   instPopulateLED.requests.row[148].pbSelection.animate := 255;
   instPopulateLED.requests.row[148].rtBackground.animate := 255;
   instPopulateLED.requests.row[148].tfDropZone.animate := 255;
   instPopulateLED.requests.row[148].tfDropZone.value := WSTRING#'';
   instPopulateLED.requests.row[148].tfLine.animate := 255;
   instPopulateLED.requests.row[148].tfLine.value := WSTRING#'';
   instPopulateLED.requests.row[148].tfPartNumber.animateDL := 255;
   instPopulateLED.requests.row[148].tfPartNumber.animateSL := 255;
   instPopulateLED.requests.row[148].tfPartNumber.value := WSTRING#'';
   instPopulateLED.requests.row[148].tfTime.animate := 255;
   instPopulateLED.requests.row[148].tfTime.value := WSTRING#'';
   instPopulateLED.requests.row[149].pbSelection.animate := 255;
   instPopulateLED.requests.row[149].rtBackground.animate := 255;
   instPopulateLED.requests.row[149].tfDropZone.animate := 255;
   instPopulateLED.requests.row[149].tfDropZone.value := WSTRING#'';
   instPopulateLED.requests.row[149].tfLine.animate := 255;
   instPopulateLED.requests.row[149].tfLine.value := WSTRING#'';
   instPopulateLED.requests.row[149].tfPartNumber.animateDL := 255;
   instPopulateLED.requests.row[149].tfPartNumber.animateSL := 255;
   instPopulateLED.requests.row[149].tfPartNumber.value := WSTRING#'';
   instPopulateLED.requests.row[149].tfTime.animate := 255;
   instPopulateLED.requests.row[149].tfTime.value := WSTRING#'';
   instPopulateLED.requests.row[150].pbSelection.animate := 255;
   instPopulateLED.requests.row[150].rtBackground.animate := 255;
   instPopulateLED.requests.row[150].tfDropZone.animate := 255;
   instPopulateLED.requests.row[150].tfDropZone.value := WSTRING#'';
   instPopulateLED.requests.row[150].tfLine.animate := 255;
   instPopulateLED.requests.row[150].tfLine.value := WSTRING#'';
   instPopulateLED.requests.row[150].tfPartNumber.animateDL := 255;
   instPopulateLED.requests.row[150].tfPartNumber.animateSL := 255;
   instPopulateLED.requests.row[150].tfPartNumber.value := WSTRING#'';
   instPopulateLED.requests.row[150].tfTime.animate := 255;
   instPopulateLED.requests.row[150].tfTime.value := WSTRING#'';
   instPopulateLED.requests.row[151].pbSelection.animate := 255;
   instPopulateLED.requests.row[151].rtBackground.animate := 255;
   instPopulateLED.requests.row[151].tfDropZone.animate := 255;
   instPopulateLED.requests.row[151].tfDropZone.value := WSTRING#'';
   instPopulateLED.requests.row[151].tfLine.animate := 255;
   instPopulateLED.requests.row[151].tfLine.value := WSTRING#'';
   instPopulateLED.requests.row[151].tfPartNumber.animateDL := 255;
   instPopulateLED.requests.row[151].tfPartNumber.animateSL := 255;
   instPopulateLED.requests.row[151].tfPartNumber.value := WSTRING#'';
   instPopulateLED.requests.row[151].tfTime.animate := 255;
   instPopulateLED.requests.row[151].tfTime.value := WSTRING#'';
   instPopulateLED.requests.row[152].pbSelection.animate := 255;
   instPopulateLED.requests.row[152].rtBackground.animate := 255;
   instPopulateLED.requests.row[152].tfDropZone.animate := 255;
   instPopulateLED.requests.row[152].tfDropZone.value := WSTRING#'';
   instPopulateLED.requests.row[152].tfLine.animate := 255;
   instPopulateLED.requests.row[152].tfLine.value := WSTRING#'';
   instPopulateLED.requests.row[152].tfPartNumber.animateDL := 255;
   instPopulateLED.requests.row[152].tfPartNumber.animateSL := 255;
   instPopulateLED.requests.row[152].tfPartNumber.value := WSTRING#'';
   instPopulateLED.requests.row[152].tfTime.animate := 255;
   instPopulateLED.requests.row[152].tfTime.value := WSTRING#'';
   instPopulateLED.requests.row[153].pbSelection.animate := 255;
   instPopulateLED.requests.row[153].rtBackground.animate := 255;
   instPopulateLED.requests.row[153].tfDropZone.animate := 255;
   instPopulateLED.requests.row[153].tfDropZone.value := WSTRING#'';
   instPopulateLED.requests.row[153].tfLine.animate := 255;
   instPopulateLED.requests.row[153].tfLine.value := WSTRING#'';
   instPopulateLED.requests.row[153].tfPartNumber.animateDL := 255;
   instPopulateLED.requests.row[153].tfPartNumber.animateSL := 255;
   instPopulateLED.requests.row[153].tfPartNumber.value := WSTRING#'';
   instPopulateLED.requests.row[153].tfTime.animate := 255;
   instPopulateLED.requests.row[153].tfTime.value := WSTRING#'';
   instPopulateLED.requests.row[154].pbSelection.animate := 255;
   instPopulateLED.requests.row[154].rtBackground.animate := 255;
   instPopulateLED.requests.row[154].tfDropZone.animate := 255;
   instPopulateLED.requests.row[154].tfDropZone.value := WSTRING#'';
   instPopulateLED.requests.row[154].tfLine.animate := 255;
   instPopulateLED.requests.row[154].tfLine.value := WSTRING#'';
   instPopulateLED.requests.row[154].tfPartNumber.animateDL := 255;
   instPopulateLED.requests.row[154].tfPartNumber.animateSL := 255;
   instPopulateLED.requests.row[154].tfPartNumber.value := WSTRING#'';
   instPopulateLED.requests.row[154].tfTime.animate := 255;
   instPopulateLED.requests.row[154].tfTime.value := WSTRING#'';
   instPopulateLED.requests.row[155].pbSelection.animate := 255;
   instPopulateLED.requests.row[155].rtBackground.animate := 255;
   instPopulateLED.requests.row[155].tfDropZone.animate := 255;
   instPopulateLED.requests.row[155].tfDropZone.value := WSTRING#'';
   instPopulateLED.requests.row[155].tfLine.animate := 255;
   instPopulateLED.requests.row[155].tfLine.value := WSTRING#'';
   instPopulateLED.requests.row[155].tfPartNumber.animateDL := 255;
   instPopulateLED.requests.row[155].tfPartNumber.animateSL := 255;
   instPopulateLED.requests.row[155].tfPartNumber.value := WSTRING#'';
   instPopulateLED.requests.row[155].tfTime.animate := 255;
   instPopulateLED.requests.row[155].tfTime.value := WSTRING#'';
   instPopulateLED.requests.row[156].pbSelection.animate := 255;
   instPopulateLED.requests.row[156].rtBackground.animate := 255;
   instPopulateLED.requests.row[156].tfDropZone.animate := 255;
   instPopulateLED.requests.row[156].tfDropZone.value := WSTRING#'';
   instPopulateLED.requests.row[156].tfLine.animate := 255;
   instPopulateLED.requests.row[156].tfLine.value := WSTRING#'';
   instPopulateLED.requests.row[156].tfPartNumber.animateDL := 255;
   instPopulateLED.requests.row[156].tfPartNumber.animateSL := 255;
   instPopulateLED.requests.row[156].tfPartNumber.value := WSTRING#'';
   instPopulateLED.requests.row[156].tfTime.animate := 255;
   instPopulateLED.requests.row[156].tfTime.value := WSTRING#'';
   instPopulateLED.requests.row[157].pbSelection.animate := 255;
   instPopulateLED.requests.row[157].rtBackground.animate := 255;
   instPopulateLED.requests.row[157].tfDropZone.animate := 255;
   instPopulateLED.requests.row[157].tfDropZone.value := WSTRING#'';
   instPopulateLED.requests.row[157].tfLine.animate := 255;
   instPopulateLED.requests.row[157].tfLine.value := WSTRING#'';
   instPopulateLED.requests.row[157].tfPartNumber.animateDL := 255;
   instPopulateLED.requests.row[157].tfPartNumber.animateSL := 255;
   instPopulateLED.requests.row[157].tfPartNumber.value := WSTRING#'';
   instPopulateLED.requests.row[157].tfTime.animate := 255;
   instPopulateLED.requests.row[157].tfTime.value := WSTRING#'';
   instPopulateLED.requests.row[158].pbSelection.animate := 255;
   instPopulateLED.requests.row[158].rtBackground.animate := 255;
   instPopulateLED.requests.row[158].tfDropZone.animate := 255;
   instPopulateLED.requests.row[158].tfDropZone.value := WSTRING#'';
   instPopulateLED.requests.row[158].tfLine.animate := 255;
   instPopulateLED.requests.row[158].tfLine.value := WSTRING#'';
   instPopulateLED.requests.row[158].tfPartNumber.animateDL := 255;
   instPopulateLED.requests.row[158].tfPartNumber.animateSL := 255;
   instPopulateLED.requests.row[158].tfPartNumber.value := WSTRING#'';
   instPopulateLED.requests.row[158].tfTime.animate := 255;
   instPopulateLED.requests.row[158].tfTime.value := WSTRING#'';
   instPopulateLED.requests.row[159].pbSelection.animate := 255;
   instPopulateLED.requests.row[159].rtBackground.animate := 255;
   instPopulateLED.requests.row[159].tfDropZone.animate := 255;
   instPopulateLED.requests.row[159].tfDropZone.value := WSTRING#'';
   instPopulateLED.requests.row[159].tfLine.animate := 255;
   instPopulateLED.requests.row[159].tfLine.value := WSTRING#'';
   instPopulateLED.requests.row[159].tfPartNumber.animateDL := 255;
   instPopulateLED.requests.row[159].tfPartNumber.animateSL := 255;
   instPopulateLED.requests.row[159].tfPartNumber.value := WSTRING#'';
   instPopulateLED.requests.row[159].tfTime.animate := 255;
   instPopulateLED.requests.row[159].tfTime.value := WSTRING#'';
   instPopulateLED.requests.row[160].pbSelection.animate := 255;
   instPopulateLED.requests.row[160].rtBackground.animate := 255;
   instPopulateLED.requests.row[160].tfDropZone.animate := 255;
   instPopulateLED.requests.row[160].tfDropZone.value := WSTRING#'';
   instPopulateLED.requests.row[160].tfLine.animate := 255;
   instPopulateLED.requests.row[160].tfLine.value := WSTRING#'';
   instPopulateLED.requests.row[160].tfPartNumber.animateDL := 255;
   instPopulateLED.requests.row[160].tfPartNumber.animateSL := 255;
   instPopulateLED.requests.row[160].tfPartNumber.value := WSTRING#'';
   instPopulateLED.requests.row[160].tfTime.animate := 255;
   instPopulateLED.requests.row[160].tfTime.value := WSTRING#'';
   instPopulateLED.requests.row[161].pbSelection.animate := 255;
   instPopulateLED.requests.row[161].rtBackground.animate := 255;
   instPopulateLED.requests.row[161].tfDropZone.animate := 255;
   instPopulateLED.requests.row[161].tfDropZone.value := WSTRING#'';
   instPopulateLED.requests.row[161].tfLine.animate := 255;
   instPopulateLED.requests.row[161].tfLine.value := WSTRING#'';
   instPopulateLED.requests.row[161].tfPartNumber.animateDL := 255;
   instPopulateLED.requests.row[161].tfPartNumber.animateSL := 255;
   instPopulateLED.requests.row[161].tfPartNumber.value := WSTRING#'';
   instPopulateLED.requests.row[161].tfTime.animate := 255;
   instPopulateLED.requests.row[161].tfTime.value := WSTRING#'';
   instPopulateLED.requests.row[162].pbSelection.animate := 255;
   instPopulateLED.requests.row[162].rtBackground.animate := 255;
   instPopulateLED.requests.row[162].tfDropZone.animate := 255;
   instPopulateLED.requests.row[162].tfDropZone.value := WSTRING#'';
   instPopulateLED.requests.row[162].tfLine.animate := 255;
   instPopulateLED.requests.row[162].tfLine.value := WSTRING#'';
   instPopulateLED.requests.row[162].tfPartNumber.animateDL := 255;
   instPopulateLED.requests.row[162].tfPartNumber.animateSL := 255;
   instPopulateLED.requests.row[162].tfPartNumber.value := WSTRING#'';
   instPopulateLED.requests.row[162].tfTime.animate := 255;
   instPopulateLED.requests.row[162].tfTime.value := WSTRING#'';
   instPopulateLED.requests.row[163].pbSelection.animate := 255;
   instPopulateLED.requests.row[163].rtBackground.animate := 255;
   instPopulateLED.requests.row[163].tfDropZone.animate := 255;
   instPopulateLED.requests.row[163].tfDropZone.value := WSTRING#'';
   instPopulateLED.requests.row[163].tfLine.animate := 255;
   instPopulateLED.requests.row[163].tfLine.value := WSTRING#'';
   instPopulateLED.requests.row[163].tfPartNumber.animateDL := 255;
   instPopulateLED.requests.row[163].tfPartNumber.animateSL := 255;
   instPopulateLED.requests.row[163].tfPartNumber.value := WSTRING#'';
   instPopulateLED.requests.row[163].tfTime.animate := 255;
   instPopulateLED.requests.row[163].tfTime.value := WSTRING#'';
   instPopulateLED.requests.row[164].pbSelection.animate := 255;
   instPopulateLED.requests.row[164].rtBackground.animate := 255;
   instPopulateLED.requests.row[164].tfDropZone.animate := 255;
   instPopulateLED.requests.row[164].tfDropZone.value := WSTRING#'';
   instPopulateLED.requests.row[164].tfLine.animate := 255;
   instPopulateLED.requests.row[164].tfLine.value := WSTRING#'';
   instPopulateLED.requests.row[164].tfPartNumber.animateDL := 255;
   instPopulateLED.requests.row[164].tfPartNumber.animateSL := 255;
   instPopulateLED.requests.row[164].tfPartNumber.value := WSTRING#'';
   instPopulateLED.requests.row[164].tfTime.animate := 255;
   instPopulateLED.requests.row[164].tfTime.value := WSTRING#'';
   instPopulateLED.requests.row[165].pbSelection.animate := 255;
   instPopulateLED.requests.row[165].rtBackground.animate := 255;
   instPopulateLED.requests.row[165].tfDropZone.animate := 255;
   instPopulateLED.requests.row[165].tfDropZone.value := WSTRING#'';
   instPopulateLED.requests.row[165].tfLine.animate := 255;
   instPopulateLED.requests.row[165].tfLine.value := WSTRING#'';
   instPopulateLED.requests.row[165].tfPartNumber.animateDL := 255;
   instPopulateLED.requests.row[165].tfPartNumber.animateSL := 255;
   instPopulateLED.requests.row[165].tfPartNumber.value := WSTRING#'';
   instPopulateLED.requests.row[165].tfTime.animate := 255;
   instPopulateLED.requests.row[165].tfTime.value := WSTRING#'';
   instPopulateLED.requests.row[166].pbSelection.animate := 255;
   instPopulateLED.requests.row[166].rtBackground.animate := 255;
   instPopulateLED.requests.row[166].tfDropZone.animate := 255;
   instPopulateLED.requests.row[166].tfDropZone.value := WSTRING#'';
   instPopulateLED.requests.row[166].tfLine.animate := 255;
   instPopulateLED.requests.row[166].tfLine.value := WSTRING#'';
   instPopulateLED.requests.row[166].tfPartNumber.animateDL := 255;
   instPopulateLED.requests.row[166].tfPartNumber.animateSL := 255;
   instPopulateLED.requests.row[166].tfPartNumber.value := WSTRING#'';
   instPopulateLED.requests.row[166].tfTime.animate := 255;
   instPopulateLED.requests.row[166].tfTime.value := WSTRING#'';
   instPopulateLED.requests.row[167].pbSelection.animate := 255;
   instPopulateLED.requests.row[167].rtBackground.animate := 255;
   instPopulateLED.requests.row[167].tfDropZone.animate := 255;
   instPopulateLED.requests.row[167].tfDropZone.value := WSTRING#'';
   instPopulateLED.requests.row[167].tfLine.animate := 255;
   instPopulateLED.requests.row[167].tfLine.value := WSTRING#'';
   instPopulateLED.requests.row[167].tfPartNumber.animateDL := 255;
   instPopulateLED.requests.row[167].tfPartNumber.animateSL := 255;
   instPopulateLED.requests.row[167].tfPartNumber.value := WSTRING#'';
   instPopulateLED.requests.row[167].tfTime.animate := 255;
   instPopulateLED.requests.row[167].tfTime.value := WSTRING#'';
   instPopulateLED.requests.row[168].pbSelection.animate := 255;
   instPopulateLED.requests.row[168].rtBackground.animate := 255;
   instPopulateLED.requests.row[168].tfDropZone.animate := 255;
   instPopulateLED.requests.row[168].tfDropZone.value := WSTRING#'';
   instPopulateLED.requests.row[168].tfLine.animate := 255;
   instPopulateLED.requests.row[168].tfLine.value := WSTRING#'';
   instPopulateLED.requests.row[168].tfPartNumber.animateDL := 255;
   instPopulateLED.requests.row[168].tfPartNumber.animateSL := 255;
   instPopulateLED.requests.row[168].tfPartNumber.value := WSTRING#'';
   instPopulateLED.requests.row[168].tfTime.animate := 255;
   instPopulateLED.requests.row[168].tfTime.value := WSTRING#'';
   instPopulateLED.requests.row[169].pbSelection.animate := 255;
   instPopulateLED.requests.row[169].rtBackground.animate := 255;
   instPopulateLED.requests.row[169].tfDropZone.animate := 255;
   instPopulateLED.requests.row[169].tfDropZone.value := WSTRING#'';
   instPopulateLED.requests.row[169].tfLine.animate := 255;
   instPopulateLED.requests.row[169].tfLine.value := WSTRING#'';
   instPopulateLED.requests.row[169].tfPartNumber.animateDL := 255;
   instPopulateLED.requests.row[169].tfPartNumber.animateSL := 255;
   instPopulateLED.requests.row[169].tfPartNumber.value := WSTRING#'';
   instPopulateLED.requests.row[169].tfTime.animate := 255;
   instPopulateLED.requests.row[169].tfTime.value := WSTRING#'';
   instPopulateLED.requests.row[170].pbSelection.animate := 255;
   instPopulateLED.requests.row[170].rtBackground.animate := 255;
   instPopulateLED.requests.row[170].tfDropZone.animate := 255;
   instPopulateLED.requests.row[170].tfDropZone.value := WSTRING#'';
   instPopulateLED.requests.row[170].tfLine.animate := 255;
   instPopulateLED.requests.row[170].tfLine.value := WSTRING#'';
   instPopulateLED.requests.row[170].tfPartNumber.animateDL := 255;
   instPopulateLED.requests.row[170].tfPartNumber.animateSL := 255;
   instPopulateLED.requests.row[170].tfPartNumber.value := WSTRING#'';
   instPopulateLED.requests.row[170].tfTime.animate := 255;
   instPopulateLED.requests.row[170].tfTime.value := WSTRING#'';
   instPopulateLED.requests.row[171].pbSelection.animate := 255;
   instPopulateLED.requests.row[171].rtBackground.animate := 255;
   instPopulateLED.requests.row[171].tfDropZone.animate := 255;
   instPopulateLED.requests.row[171].tfDropZone.value := WSTRING#'';
   instPopulateLED.requests.row[171].tfLine.animate := 255;
   instPopulateLED.requests.row[171].tfLine.value := WSTRING#'';
   instPopulateLED.requests.row[171].tfPartNumber.animateDL := 255;
   instPopulateLED.requests.row[171].tfPartNumber.animateSL := 255;
   instPopulateLED.requests.row[171].tfPartNumber.value := WSTRING#'';
   instPopulateLED.requests.row[171].tfTime.animate := 255;
   instPopulateLED.requests.row[171].tfTime.value := WSTRING#'';
   instPopulateLED.requests.row[172].pbSelection.animate := 255;
   instPopulateLED.requests.row[172].rtBackground.animate := 255;
   instPopulateLED.requests.row[172].tfDropZone.animate := 255;
   instPopulateLED.requests.row[172].tfDropZone.value := WSTRING#'';
   instPopulateLED.requests.row[172].tfLine.animate := 255;
   instPopulateLED.requests.row[172].tfLine.value := WSTRING#'';
   instPopulateLED.requests.row[172].tfPartNumber.animateDL := 255;
   instPopulateLED.requests.row[172].tfPartNumber.animateSL := 255;
   instPopulateLED.requests.row[172].tfPartNumber.value := WSTRING#'';
   instPopulateLED.requests.row[172].tfTime.animate := 255;
   instPopulateLED.requests.row[172].tfTime.value := WSTRING#'';
   instPopulateLED.requests.row[173].pbSelection.animate := 255;
   instPopulateLED.requests.row[173].rtBackground.animate := 255;
   instPopulateLED.requests.row[173].tfDropZone.animate := 255;
   instPopulateLED.requests.row[173].tfDropZone.value := WSTRING#'';
   instPopulateLED.requests.row[173].tfLine.animate := 255;
   instPopulateLED.requests.row[173].tfLine.value := WSTRING#'';
   instPopulateLED.requests.row[173].tfPartNumber.animateDL := 255;
   instPopulateLED.requests.row[173].tfPartNumber.animateSL := 255;
   instPopulateLED.requests.row[173].tfPartNumber.value := WSTRING#'';
   instPopulateLED.requests.row[173].tfTime.animate := 255;
   instPopulateLED.requests.row[173].tfTime.value := WSTRING#'';
   instPopulateLED.requests.row[174].pbSelection.animate := 255;
   instPopulateLED.requests.row[174].rtBackground.animate := 255;
   instPopulateLED.requests.row[174].tfDropZone.animate := 255;
   instPopulateLED.requests.row[174].tfDropZone.value := WSTRING#'';
   instPopulateLED.requests.row[174].tfLine.animate := 255;
   instPopulateLED.requests.row[174].tfLine.value := WSTRING#'';
   instPopulateLED.requests.row[174].tfPartNumber.animateDL := 255;
   instPopulateLED.requests.row[174].tfPartNumber.animateSL := 255;
   instPopulateLED.requests.row[174].tfPartNumber.value := WSTRING#'';
   instPopulateLED.requests.row[174].tfTime.animate := 255;
   instPopulateLED.requests.row[174].tfTime.value := WSTRING#'';
   instPopulateLED.requests.row[175].pbSelection.animate := 255;
   instPopulateLED.requests.row[175].rtBackground.animate := 255;
   instPopulateLED.requests.row[175].tfDropZone.animate := 255;
   instPopulateLED.requests.row[175].tfDropZone.value := WSTRING#'';
   instPopulateLED.requests.row[175].tfLine.animate := 255;
   instPopulateLED.requests.row[175].tfLine.value := WSTRING#'';
   instPopulateLED.requests.row[175].tfPartNumber.animateDL := 255;
   instPopulateLED.requests.row[175].tfPartNumber.animateSL := 255;
   instPopulateLED.requests.row[175].tfPartNumber.value := WSTRING#'';
   instPopulateLED.requests.row[175].tfTime.animate := 255;
   instPopulateLED.requests.row[175].tfTime.value := WSTRING#'';
   instPopulateLED.requests.row[176].pbSelection.animate := 255;
   instPopulateLED.requests.row[176].rtBackground.animate := 255;
   instPopulateLED.requests.row[176].tfDropZone.animate := 255;
   instPopulateLED.requests.row[176].tfDropZone.value := WSTRING#'';
   instPopulateLED.requests.row[176].tfLine.animate := 255;
   instPopulateLED.requests.row[176].tfLine.value := WSTRING#'';
   instPopulateLED.requests.row[176].tfPartNumber.animateDL := 255;
   instPopulateLED.requests.row[176].tfPartNumber.animateSL := 255;
   instPopulateLED.requests.row[176].tfPartNumber.value := WSTRING#'';
   instPopulateLED.requests.row[176].tfTime.animate := 255;
   instPopulateLED.requests.row[176].tfTime.value := WSTRING#'';
   instPopulateLED.requests.row[177].pbSelection.animate := 255;
   instPopulateLED.requests.row[177].rtBackground.animate := 255;
   instPopulateLED.requests.row[177].tfDropZone.animate := 255;
   instPopulateLED.requests.row[177].tfDropZone.value := WSTRING#'';
   instPopulateLED.requests.row[177].tfLine.animate := 255;
   instPopulateLED.requests.row[177].tfLine.value := WSTRING#'';
   instPopulateLED.requests.row[177].tfPartNumber.animateDL := 255;
   instPopulateLED.requests.row[177].tfPartNumber.animateSL := 255;
   instPopulateLED.requests.row[177].tfPartNumber.value := WSTRING#'';
   instPopulateLED.requests.row[177].tfTime.animate := 255;
   instPopulateLED.requests.row[177].tfTime.value := WSTRING#'';
   instPopulateLED.requests.row[178].pbSelection.animate := 255;
   instPopulateLED.requests.row[178].rtBackground.animate := 255;
   instPopulateLED.requests.row[178].tfDropZone.animate := 255;
   instPopulateLED.requests.row[178].tfDropZone.value := WSTRING#'';
   instPopulateLED.requests.row[178].tfLine.animate := 255;
   instPopulateLED.requests.row[178].tfLine.value := WSTRING#'';
   instPopulateLED.requests.row[178].tfPartNumber.animateDL := 255;
   instPopulateLED.requests.row[178].tfPartNumber.animateSL := 255;
   instPopulateLED.requests.row[178].tfPartNumber.value := WSTRING#'';
   instPopulateLED.requests.row[178].tfTime.animate := 255;
   instPopulateLED.requests.row[178].tfTime.value := WSTRING#'';
   instPopulateLED.requests.row[179].pbSelection.animate := 255;
   instPopulateLED.requests.row[179].rtBackground.animate := 255;
   instPopulateLED.requests.row[179].tfDropZone.animate := 255;
   instPopulateLED.requests.row[179].tfDropZone.value := WSTRING#'';
   instPopulateLED.requests.row[179].tfLine.animate := 255;
   instPopulateLED.requests.row[179].tfLine.value := WSTRING#'';
   instPopulateLED.requests.row[179].tfPartNumber.animateDL := 255;
   instPopulateLED.requests.row[179].tfPartNumber.animateSL := 255;
   instPopulateLED.requests.row[179].tfPartNumber.value := WSTRING#'';
   instPopulateLED.requests.row[179].tfTime.animate := 255;
   instPopulateLED.requests.row[179].tfTime.value := WSTRING#'';
   instPopulateLED.requests.row[180].pbSelection.animate := 255;
   instPopulateLED.requests.row[180].rtBackground.animate := 255;
   instPopulateLED.requests.row[180].tfDropZone.animate := 255;
   instPopulateLED.requests.row[180].tfDropZone.value := WSTRING#'';
   instPopulateLED.requests.row[180].tfLine.animate := 255;
   instPopulateLED.requests.row[180].tfLine.value := WSTRING#'';
   instPopulateLED.requests.row[180].tfPartNumber.animateDL := 255;
   instPopulateLED.requests.row[180].tfPartNumber.animateSL := 255;
   instPopulateLED.requests.row[180].tfPartNumber.value := WSTRING#'';
   instPopulateLED.requests.row[180].tfTime.animate := 255;
   instPopulateLED.requests.row[180].tfTime.value := WSTRING#'';
   instPopulateLED.requests.row[181].pbSelection.animate := 255;
   instPopulateLED.requests.row[181].rtBackground.animate := 255;
   instPopulateLED.requests.row[181].tfDropZone.animate := 255;
   instPopulateLED.requests.row[181].tfDropZone.value := WSTRING#'';
   instPopulateLED.requests.row[181].tfLine.animate := 255;
   instPopulateLED.requests.row[181].tfLine.value := WSTRING#'';
   instPopulateLED.requests.row[181].tfPartNumber.animateDL := 255;
   instPopulateLED.requests.row[181].tfPartNumber.animateSL := 255;
   instPopulateLED.requests.row[181].tfPartNumber.value := WSTRING#'';
   instPopulateLED.requests.row[181].tfTime.animate := 255;
   instPopulateLED.requests.row[181].tfTime.value := WSTRING#'';
   instPopulateLED.requests.row[182].pbSelection.animate := 255;
   instPopulateLED.requests.row[182].rtBackground.animate := 255;
   instPopulateLED.requests.row[182].tfDropZone.animate := 255;
   instPopulateLED.requests.row[182].tfDropZone.value := WSTRING#'';
   instPopulateLED.requests.row[182].tfLine.animate := 255;
   instPopulateLED.requests.row[182].tfLine.value := WSTRING#'';
   instPopulateLED.requests.row[182].tfPartNumber.animateDL := 255;
   instPopulateLED.requests.row[182].tfPartNumber.animateSL := 255;
   instPopulateLED.requests.row[182].tfPartNumber.value := WSTRING#'';
   instPopulateLED.requests.row[182].tfTime.animate := 255;
   instPopulateLED.requests.row[182].tfTime.value := WSTRING#'';
   instPopulateLED.requests.row[183].pbSelection.animate := 255;
   instPopulateLED.requests.row[183].rtBackground.animate := 255;
   instPopulateLED.requests.row[183].tfDropZone.animate := 255;
   instPopulateLED.requests.row[183].tfDropZone.value := WSTRING#'';
   instPopulateLED.requests.row[183].tfLine.animate := 255;
   instPopulateLED.requests.row[183].tfLine.value := WSTRING#'';
   instPopulateLED.requests.row[183].tfPartNumber.animateDL := 255;
   instPopulateLED.requests.row[183].tfPartNumber.animateSL := 255;
   instPopulateLED.requests.row[183].tfPartNumber.value := WSTRING#'';
   instPopulateLED.requests.row[183].tfTime.animate := 255;
   instPopulateLED.requests.row[183].tfTime.value := WSTRING#'';
   instPopulateLED.requests.row[184].pbSelection.animate := 255;
   instPopulateLED.requests.row[184].rtBackground.animate := 255;
   instPopulateLED.requests.row[184].tfDropZone.animate := 255;
   instPopulateLED.requests.row[184].tfDropZone.value := WSTRING#'';
   instPopulateLED.requests.row[184].tfLine.animate := 255;
   instPopulateLED.requests.row[184].tfLine.value := WSTRING#'';
   instPopulateLED.requests.row[184].tfPartNumber.animateDL := 255;
   instPopulateLED.requests.row[184].tfPartNumber.animateSL := 255;
   instPopulateLED.requests.row[184].tfPartNumber.value := WSTRING#'';
   instPopulateLED.requests.row[184].tfTime.animate := 255;
   instPopulateLED.requests.row[184].tfTime.value := WSTRING#'';
   instPopulateLED.requests.row[185].pbSelection.animate := 255;
   instPopulateLED.requests.row[185].rtBackground.animate := 255;
   instPopulateLED.requests.row[185].tfDropZone.animate := 255;
   instPopulateLED.requests.row[185].tfDropZone.value := WSTRING#'';
   instPopulateLED.requests.row[185].tfLine.animate := 255;
   instPopulateLED.requests.row[185].tfLine.value := WSTRING#'';
   instPopulateLED.requests.row[185].tfPartNumber.animateDL := 255;
   instPopulateLED.requests.row[185].tfPartNumber.animateSL := 255;
   instPopulateLED.requests.row[185].tfPartNumber.value := WSTRING#'';
   instPopulateLED.requests.row[185].tfTime.animate := 255;
   instPopulateLED.requests.row[185].tfTime.value := WSTRING#'';
   instPopulateLED.requests.row[186].pbSelection.animate := 255;
   instPopulateLED.requests.row[186].rtBackground.animate := 255;
   instPopulateLED.requests.row[186].tfDropZone.animate := 255;
   instPopulateLED.requests.row[186].tfDropZone.value := WSTRING#'';
   instPopulateLED.requests.row[186].tfLine.animate := 255;
   instPopulateLED.requests.row[186].tfLine.value := WSTRING#'';
   instPopulateLED.requests.row[186].tfPartNumber.animateDL := 255;
   instPopulateLED.requests.row[186].tfPartNumber.animateSL := 255;
   instPopulateLED.requests.row[186].tfPartNumber.value := WSTRING#'';
   instPopulateLED.requests.row[186].tfTime.animate := 255;
   instPopulateLED.requests.row[186].tfTime.value := WSTRING#'';
   instPopulateLED.requests.row[187].pbSelection.animate := 255;
   instPopulateLED.requests.row[187].rtBackground.animate := 255;
   instPopulateLED.requests.row[187].tfDropZone.animate := 255;
   instPopulateLED.requests.row[187].tfDropZone.value := WSTRING#'';
   instPopulateLED.requests.row[187].tfLine.animate := 255;
   instPopulateLED.requests.row[187].tfLine.value := WSTRING#'';
   instPopulateLED.requests.row[187].tfPartNumber.animateDL := 255;
   instPopulateLED.requests.row[187].tfPartNumber.animateSL := 255;
   instPopulateLED.requests.row[187].tfPartNumber.value := WSTRING#'';
   instPopulateLED.requests.row[187].tfTime.animate := 255;
   instPopulateLED.requests.row[187].tfTime.value := WSTRING#'';
   instPopulateLED.requests.row[188].pbSelection.animate := 255;
   instPopulateLED.requests.row[188].rtBackground.animate := 255;
   instPopulateLED.requests.row[188].tfDropZone.animate := 255;
   instPopulateLED.requests.row[188].tfDropZone.value := WSTRING#'';
   instPopulateLED.requests.row[188].tfLine.animate := 255;
   instPopulateLED.requests.row[188].tfLine.value := WSTRING#'';
   instPopulateLED.requests.row[188].tfPartNumber.animateDL := 255;
   instPopulateLED.requests.row[188].tfPartNumber.animateSL := 255;
   instPopulateLED.requests.row[188].tfPartNumber.value := WSTRING#'';
   instPopulateLED.requests.row[188].tfTime.animate := 255;
   instPopulateLED.requests.row[188].tfTime.value := WSTRING#'';
   instPopulateLED.requests.row[189].pbSelection.animate := 255;
   instPopulateLED.requests.row[189].rtBackground.animate := 255;
   instPopulateLED.requests.row[189].tfDropZone.animate := 255;
   instPopulateLED.requests.row[189].tfDropZone.value := WSTRING#'';
   instPopulateLED.requests.row[189].tfLine.animate := 255;
   instPopulateLED.requests.row[189].tfLine.value := WSTRING#'';
   instPopulateLED.requests.row[189].tfPartNumber.animateDL := 255;
   instPopulateLED.requests.row[189].tfPartNumber.animateSL := 255;
   instPopulateLED.requests.row[189].tfPartNumber.value := WSTRING#'';
   instPopulateLED.requests.row[189].tfTime.animate := 255;
   instPopulateLED.requests.row[189].tfTime.value := WSTRING#'';
   instPopulateLED.requests.row[190].pbSelection.animate := 255;
   instPopulateLED.requests.row[190].rtBackground.animate := 255;
   instPopulateLED.requests.row[190].tfDropZone.animate := 255;
   instPopulateLED.requests.row[190].tfDropZone.value := WSTRING#'';
   instPopulateLED.requests.row[190].tfLine.animate := 255;
   instPopulateLED.requests.row[190].tfLine.value := WSTRING#'';
   instPopulateLED.requests.row[190].tfPartNumber.animateDL := 255;
   instPopulateLED.requests.row[190].tfPartNumber.animateSL := 255;
   instPopulateLED.requests.row[190].tfPartNumber.value := WSTRING#'';
   instPopulateLED.requests.row[190].tfTime.animate := 255;
   instPopulateLED.requests.row[190].tfTime.value := WSTRING#'';
   instPopulateLED.requests.row[191].pbSelection.animate := 255;
   instPopulateLED.requests.row[191].rtBackground.animate := 255;
   instPopulateLED.requests.row[191].tfDropZone.animate := 255;
   instPopulateLED.requests.row[191].tfDropZone.value := WSTRING#'';
   instPopulateLED.requests.row[191].tfLine.animate := 255;
   instPopulateLED.requests.row[191].tfLine.value := WSTRING#'';
   instPopulateLED.requests.row[191].tfPartNumber.animateDL := 255;
   instPopulateLED.requests.row[191].tfPartNumber.animateSL := 255;
   instPopulateLED.requests.row[191].tfPartNumber.value := WSTRING#'';
   instPopulateLED.requests.row[191].tfTime.animate := 255;
   instPopulateLED.requests.row[191].tfTime.value := WSTRING#'';
   instPopulateLED.requests.row[192].pbSelection.animate := 255;
   instPopulateLED.requests.row[192].rtBackground.animate := 255;
   instPopulateLED.requests.row[192].tfDropZone.animate := 255;
   instPopulateLED.requests.row[192].tfDropZone.value := WSTRING#'';
   instPopulateLED.requests.row[192].tfLine.animate := 255;
   instPopulateLED.requests.row[192].tfLine.value := WSTRING#'';
   instPopulateLED.requests.row[192].tfPartNumber.animateDL := 255;
   instPopulateLED.requests.row[192].tfPartNumber.animateSL := 255;
   instPopulateLED.requests.row[192].tfPartNumber.value := WSTRING#'';
   instPopulateLED.requests.row[192].tfTime.animate := 255;
   instPopulateLED.requests.row[192].tfTime.value := WSTRING#'';
   instPopulateLED.requests.row[193].pbSelection.animate := 255;
   instPopulateLED.requests.row[193].rtBackground.animate := 255;
   instPopulateLED.requests.row[193].tfDropZone.animate := 255;
   instPopulateLED.requests.row[193].tfDropZone.value := WSTRING#'';
   instPopulateLED.requests.row[193].tfLine.animate := 255;
   instPopulateLED.requests.row[193].tfLine.value := WSTRING#'';
   instPopulateLED.requests.row[193].tfPartNumber.animateDL := 255;
   instPopulateLED.requests.row[193].tfPartNumber.animateSL := 255;
   instPopulateLED.requests.row[193].tfPartNumber.value := WSTRING#'';
   instPopulateLED.requests.row[193].tfTime.animate := 255;
   instPopulateLED.requests.row[193].tfTime.value := WSTRING#'';
   instPopulateLED.requests.row[194].pbSelection.animate := 255;
   instPopulateLED.requests.row[194].rtBackground.animate := 255;
   instPopulateLED.requests.row[194].tfDropZone.animate := 255;
   instPopulateLED.requests.row[194].tfDropZone.value := WSTRING#'';
   instPopulateLED.requests.row[194].tfLine.animate := 255;
   instPopulateLED.requests.row[194].tfLine.value := WSTRING#'';
   instPopulateLED.requests.row[194].tfPartNumber.animateDL := 255;
   instPopulateLED.requests.row[194].tfPartNumber.animateSL := 255;
   instPopulateLED.requests.row[194].tfPartNumber.value := WSTRING#'';
   instPopulateLED.requests.row[194].tfTime.animate := 255;
   instPopulateLED.requests.row[194].tfTime.value := WSTRING#'';
   instPopulateLED.requests.row[195].pbSelection.animate := 255;
   instPopulateLED.requests.row[195].rtBackground.animate := 255;
   instPopulateLED.requests.row[195].tfDropZone.animate := 255;
   instPopulateLED.requests.row[195].tfDropZone.value := WSTRING#'';
   instPopulateLED.requests.row[195].tfLine.animate := 255;
   instPopulateLED.requests.row[195].tfLine.value := WSTRING#'';
   instPopulateLED.requests.row[195].tfPartNumber.animateDL := 255;
   instPopulateLED.requests.row[195].tfPartNumber.animateSL := 255;
   instPopulateLED.requests.row[195].tfPartNumber.value := WSTRING#'';
   instPopulateLED.requests.row[195].tfTime.animate := 255;
   instPopulateLED.requests.row[195].tfTime.value := WSTRING#'';
   instPopulateLED.requests.row[196].pbSelection.animate := 255;
   instPopulateLED.requests.row[196].rtBackground.animate := 255;
   instPopulateLED.requests.row[196].tfDropZone.animate := 255;
   instPopulateLED.requests.row[196].tfDropZone.value := WSTRING#'';
   instPopulateLED.requests.row[196].tfLine.animate := 255;
   instPopulateLED.requests.row[196].tfLine.value := WSTRING#'';
   instPopulateLED.requests.row[196].tfPartNumber.animateDL := 255;
   instPopulateLED.requests.row[196].tfPartNumber.animateSL := 255;
   instPopulateLED.requests.row[196].tfPartNumber.value := WSTRING#'';
   instPopulateLED.requests.row[196].tfTime.animate := 255;
   instPopulateLED.requests.row[196].tfTime.value := WSTRING#'';
   instPopulateLED.requests.row[197].pbSelection.animate := 255;
   instPopulateLED.requests.row[197].rtBackground.animate := 255;
   instPopulateLED.requests.row[197].tfDropZone.animate := 255;
   instPopulateLED.requests.row[197].tfDropZone.value := WSTRING#'';
   instPopulateLED.requests.row[197].tfLine.animate := 255;
   instPopulateLED.requests.row[197].tfLine.value := WSTRING#'';
   instPopulateLED.requests.row[197].tfPartNumber.animateDL := 255;
   instPopulateLED.requests.row[197].tfPartNumber.animateSL := 255;
   instPopulateLED.requests.row[197].tfPartNumber.value := WSTRING#'';
   instPopulateLED.requests.row[197].tfTime.animate := 255;
   instPopulateLED.requests.row[197].tfTime.value := WSTRING#'';
   instPopulateLED.requests.row[198].pbSelection.animate := 255;
   instPopulateLED.requests.row[198].rtBackground.animate := 255;
   instPopulateLED.requests.row[198].tfDropZone.animate := 255;
   instPopulateLED.requests.row[198].tfDropZone.value := WSTRING#'';
   instPopulateLED.requests.row[198].tfLine.animate := 255;
   instPopulateLED.requests.row[198].tfLine.value := WSTRING#'';
   instPopulateLED.requests.row[198].tfPartNumber.animateDL := 255;
   instPopulateLED.requests.row[198].tfPartNumber.animateSL := 255;
   instPopulateLED.requests.row[198].tfPartNumber.value := WSTRING#'';
   instPopulateLED.requests.row[198].tfTime.animate := 255;
   instPopulateLED.requests.row[198].tfTime.value := WSTRING#'';
   instPopulateLED.requests.row[199].pbSelection.animate := 255;
   instPopulateLED.requests.row[199].rtBackground.animate := 255;
   instPopulateLED.requests.row[199].tfDropZone.animate := 255;
   instPopulateLED.requests.row[199].tfDropZone.value := WSTRING#'';
   instPopulateLED.requests.row[199].tfLine.animate := 255;
   instPopulateLED.requests.row[199].tfLine.value := WSTRING#'';
   instPopulateLED.requests.row[199].tfPartNumber.animateDL := 255;
   instPopulateLED.requests.row[199].tfPartNumber.animateSL := 255;
   instPopulateLED.requests.row[199].tfPartNumber.value := WSTRING#'';
   instPopulateLED.requests.row[199].tfTime.animate := 255;
   instPopulateLED.requests.row[199].tfTime.value := WSTRING#'';
   instRcrdPartReq.pRow := 6;
   instRcrdPartReq.old.presses.me[26,3] := TRUE;
   instRmvPartReq.pRow := 6;
   instRmvPartReq.old.partReq.me[26,3] := TRUE;
   stations.me[0].kp8Config.activate[3] := TRUE;
   stations.me[0].kp8Config.activate[7] := TRUE;
   stations.me[0].kp8Config.colorOn1[0] := 'off';
   stations.me[0].kp8Config.colorOn1[1] := 'off';
   stations.me[0].kp8Config.colorOn1[2] := 'off';
   stations.me[0].kp8Config.colorOn1[3] := 'yellow';
   stations.me[0].kp8Config.colorOn1[4] := 'off';
   stations.me[0].kp8Config.colorOn1[5] := 'off';
   stations.me[0].kp8Config.colorOn1[6] := 'off';
   stations.me[0].kp8Config.colorOn1[7] := 'yellow';
   stations.me[0].kp8Config.colorOn2[0] := 'off';
   stations.me[0].kp8Config.colorOn2[1] := 'off';
   stations.me[0].kp8Config.colorOn2[2] := 'off';
   stations.me[0].kp8Config.colorOn2[4] := 'off';
   stations.me[0].kp8Config.colorOn2[5] := 'off';
   stations.me[0].kp8Config.colorOn2[6] := 'off';
   stations.me[0].kp8Config.colorOff[0] := 'off';
   stations.me[0].kp8Config.colorOff[1] := 'off';
   stations.me[0].kp8Config.colorOff[2] := 'off';
   stations.me[0].kp8Config.colorOff[3] := 'green';
   stations.me[0].kp8Config.colorOff[4] := 'off';
   stations.me[0].kp8Config.colorOff[5] := 'off';
   stations.me[0].kp8Config.colorOff[6] := 'off';
   stations.me[0].kp8Config.colorOff[7] := 'green';
   stations.me[0].kp8Config.mode[3] := TRUE;
   stations.me[0].kp8Config.mode[7] := TRUE;
   stations.me[0].kp8Out := 16#0088_0000;
   stations.me[0].presetTime.allotted[3] := 1800.0;
   stations.me[0].presetTime.allotted[7] := 1800.0;
   stations.me[0].presetTime.critical[3] := 300.0;
   stations.me[0].presetTime.critical[7] := 300.0;
   stations.me[0].stackLightOut := 16#2400_0000;
   stations.me[1].kp8Config.activate[2] := TRUE;
   stations.me[1].kp8Config.activate[3] := TRUE;
   stations.me[1].kp8Config.activate[6] := TRUE;
   stations.me[1].kp8Config.activate[7] := TRUE;
   stations.me[1].kp8Config.colorOn1[0] := 'off';
   stations.me[1].kp8Config.colorOn1[1] := 'off';
   stations.me[1].kp8Config.colorOn1[2] := 'yellow';
   stations.me[1].kp8Config.colorOn1[3] := 'yellow';
   stations.me[1].kp8Config.colorOn1[4] := 'off';
   stations.me[1].kp8Config.colorOn1[5] := 'off';
   stations.me[1].kp8Config.colorOn1[6] := 'yellow';
   stations.me[1].kp8Config.colorOn1[7] := 'yellow';
   stations.me[1].kp8Config.colorOn2[0] := 'off';
   stations.me[1].kp8Config.colorOn2[1] := 'off';
   stations.me[1].kp8Config.colorOn2[4] := 'off';
   stations.me[1].kp8Config.colorOn2[5] := 'off';
   stations.me[1].kp8Config.colorOff[0] := 'off';
   stations.me[1].kp8Config.colorOff[1] := 'off';
   stations.me[1].kp8Config.colorOff[2] := 'green';
   stations.me[1].kp8Config.colorOff[3] := 'green';
   stations.me[1].kp8Config.colorOff[4] := 'off';
   stations.me[1].kp8Config.colorOff[5] := 'off';
   stations.me[1].kp8Config.colorOff[6] := 'green';
   stations.me[1].kp8Config.colorOff[7] := 'green';
   stations.me[1].kp8Config.mode[2] := TRUE;
   stations.me[1].kp8Config.mode[3] := TRUE;
   stations.me[1].kp8Config.mode[6] := TRUE;
   stations.me[1].kp8Config.mode[7] := TRUE;
   stations.me[1].kp8Out := 16#00CC_0000;
   stations.me[1].presetTime.allotted[2] := 1800.0;
   stations.me[1].presetTime.allotted[3] := 1800.0;
   stations.me[1].presetTime.allotted[6] := 1800.0;
   stations.me[1].presetTime.allotted[7] := 1800.0;
   stations.me[1].presetTime.critical[2] := 300.0;
   stations.me[1].presetTime.critical[3] := 300.0;
   stations.me[1].presetTime.critical[6] := 300.0;
   stations.me[1].presetTime.critical[7] := 300.0;
   stations.me[1].stackLightOut := 16#2409_0000;
   stations.me[2].kp8Config.activate[1] := TRUE;
   stations.me[2].kp8Config.activate[2] := TRUE;
   stations.me[2].kp8Config.activate[3] := TRUE;
   stations.me[2].kp8Config.activate[5] := TRUE;
   stations.me[2].kp8Config.activate[6] := TRUE;
   stations.me[2].kp8Config.activate[7] := TRUE;
   stations.me[2].kp8Config.colorOn1[0] := 'off';
   stations.me[2].kp8Config.colorOn1[1] := 'yellow';
   stations.me[2].kp8Config.colorOn1[2] := 'yellow';
   stations.me[2].kp8Config.colorOn1[3] := 'yellow';
   stations.me[2].kp8Config.colorOn1[4] := 'off';
   stations.me[2].kp8Config.colorOn1[5] := 'yellow';
   stations.me[2].kp8Config.colorOn1[6] := 'yellow';
   stations.me[2].kp8Config.colorOn1[7] := 'yellow';
   stations.me[2].kp8Config.colorOn2[0] := 'off';
   stations.me[2].kp8Config.colorOn2[4] := 'off';
   stations.me[2].kp8Config.colorOff[0] := 'off';
   stations.me[2].kp8Config.colorOff[1] := 'green';
   stations.me[2].kp8Config.colorOff[2] := 'green';
   stations.me[2].kp8Config.colorOff[3] := 'green';
   stations.me[2].kp8Config.colorOff[4] := 'off';
   stations.me[2].kp8Config.colorOff[5] := 'green';
   stations.me[2].kp8Config.colorOff[6] := 'green';
   stations.me[2].kp8Config.colorOff[7] := 'green';
   stations.me[2].kp8Config.mode[1] := TRUE;
   stations.me[2].kp8Config.mode[2] := TRUE;
   stations.me[2].kp8Config.mode[3] := TRUE;
   stations.me[2].kp8Config.mode[5] := TRUE;
   stations.me[2].kp8Config.mode[6] := TRUE;
   stations.me[2].kp8Config.mode[7] := TRUE;
   stations.me[2].kp8Out := 16#00EE_0000;
   stations.me[2].presetTime.allotted[1] := 1800.0;
   stations.me[2].presetTime.allotted[2] := 1800.0;
   stations.me[2].presetTime.allotted[3] := 1800.0;
   stations.me[2].presetTime.allotted[5] := 1800.0;
   stations.me[2].presetTime.allotted[6] := 1800.0;
   stations.me[2].presetTime.allotted[7] := 1800.0;
   stations.me[2].presetTime.critical[1] := 300.0;
   stations.me[2].presetTime.critical[2] := 300.0;
   stations.me[2].presetTime.critical[3] := 300.0;
   stations.me[2].presetTime.critical[5] := 300.0;
   stations.me[2].presetTime.critical[6] := 300.0;
   stations.me[2].presetTime.critical[7] := 300.0;
   stations.me[2].stackLightOut := 16#2449_0200;
   stations.me[3].kp8Config.activate[1] := TRUE;
   stations.me[3].kp8Config.activate[2] := TRUE;
   stations.me[3].kp8Config.activate[3] := TRUE;
   stations.me[3].kp8Config.activate[5] := TRUE;
   stations.me[3].kp8Config.activate[6] := TRUE;
   stations.me[3].kp8Config.activate[7] := TRUE;
   stations.me[3].kp8Config.colorOn1[0] := 'off';
   stations.me[3].kp8Config.colorOn1[1] := 'yellow';
   stations.me[3].kp8Config.colorOn1[2] := 'yellow';
   stations.me[3].kp8Config.colorOn1[3] := 'yellow';
   stations.me[3].kp8Config.colorOn1[4] := 'off';
   stations.me[3].kp8Config.colorOn1[5] := 'yellow';
   stations.me[3].kp8Config.colorOn1[6] := 'yellow';
   stations.me[3].kp8Config.colorOn1[7] := 'yellow';
   stations.me[3].kp8Config.colorOn2[0] := 'off';
   stations.me[3].kp8Config.colorOn2[4] := 'off';
   stations.me[3].kp8Config.colorOff[0] := 'off';
   stations.me[3].kp8Config.colorOff[1] := 'green';
   stations.me[3].kp8Config.colorOff[2] := 'green';
   stations.me[3].kp8Config.colorOff[3] := 'green';
   stations.me[3].kp8Config.colorOff[4] := 'off';
   stations.me[3].kp8Config.colorOff[5] := 'green';
   stations.me[3].kp8Config.colorOff[6] := 'green';
   stations.me[3].kp8Config.colorOff[7] := 'green';
   stations.me[3].kp8Config.mode[1] := TRUE;
   stations.me[3].kp8Config.mode[2] := TRUE;
   stations.me[3].kp8Config.mode[3] := TRUE;
   stations.me[3].kp8Config.mode[5] := TRUE;
   stations.me[3].kp8Config.mode[6] := TRUE;
   stations.me[3].kp8Config.mode[7] := TRUE;
   stations.me[3].kp8Out := 16#00EE_0000;
   stations.me[3].presetTime.allotted[1] := 1800.0;
   stations.me[3].presetTime.allotted[2] := 1800.0;
   stations.me[3].presetTime.allotted[3] := 1800.0;
   stations.me[3].presetTime.allotted[5] := 1800.0;
   stations.me[3].presetTime.allotted[6] := 1800.0;
   stations.me[3].presetTime.allotted[7] := 1800.0;
   stations.me[3].presetTime.critical[1] := 300.0;
   stations.me[3].presetTime.critical[2] := 300.0;
   stations.me[3].presetTime.critical[3] := 300.0;
   stations.me[3].presetTime.critical[5] := 300.0;
   stations.me[3].presetTime.critical[6] := 300.0;
   stations.me[3].presetTime.critical[7] := 300.0;
   stations.me[3].stackLightOut := 16#2449_0200;
   stations.me[4].kp8Config.activate[7] := TRUE;
   stations.me[4].kp8Config.colorOn1[0] := 'off';
   stations.me[4].kp8Config.colorOn1[1] := 'off';
   stations.me[4].kp8Config.colorOn1[2] := 'off';
   stations.me[4].kp8Config.colorOn1[3] := 'off';
   stations.me[4].kp8Config.colorOn1[4] := 'off';
   stations.me[4].kp8Config.colorOn1[5] := 'off';
   stations.me[4].kp8Config.colorOn1[6] := 'off';
   stations.me[4].kp8Config.colorOn1[7] := 'yellow';
   stations.me[4].kp8Config.colorOn2[0] := 'off';
   stations.me[4].kp8Config.colorOn2[1] := 'off';
   stations.me[4].kp8Config.colorOn2[2] := 'off';
   stations.me[4].kp8Config.colorOn2[3] := 'off';
   stations.me[4].kp8Config.colorOn2[4] := 'off';
   stations.me[4].kp8Config.colorOn2[5] := 'off';
   stations.me[4].kp8Config.colorOn2[6] := 'off';
   stations.me[4].kp8Config.colorOff[0] := 'off';
   stations.me[4].kp8Config.colorOff[1] := 'off';
   stations.me[4].kp8Config.colorOff[2] := 'off';
   stations.me[4].kp8Config.colorOff[3] := 'off';
   stations.me[4].kp8Config.colorOff[4] := 'off';
   stations.me[4].kp8Config.colorOff[5] := 'off';
   stations.me[4].kp8Config.colorOff[6] := 'off';
   stations.me[4].kp8Config.colorOff[7] := 'green';
   stations.me[4].kp8Config.mode[7] := TRUE;
   stations.me[4].kp8Out := 16#0080_0000;
   stations.me[4].presetTime.allotted[7] := 1800.0;
   stations.me[4].presetTime.critical[7] := 300.0;
   stations.me[4].stackLightOut := 16#0400_0000;
   stations.me[5].kp8Config.activate[1] := TRUE;
   stations.me[5].kp8Config.activate[2] := TRUE;
   stations.me[5].kp8Config.activate[3] := TRUE;
   stations.me[5].kp8Config.activate[5] := TRUE;
   stations.me[5].kp8Config.activate[6] := TRUE;
   stations.me[5].kp8Config.activate[7] := TRUE;
   stations.me[5].kp8Config.colorOn1[0] := 'off';
   stations.me[5].kp8Config.colorOn1[1] := 'yellow';
   stations.me[5].kp8Config.colorOn1[2] := 'yellow';
   stations.me[5].kp8Config.colorOn1[3] := 'yellow';
   stations.me[5].kp8Config.colorOn1[4] := 'off';
   stations.me[5].kp8Config.colorOn1[5] := 'yellow';
   stations.me[5].kp8Config.colorOn1[6] := 'yellow';
   stations.me[5].kp8Config.colorOn1[7] := 'yellow';
   stations.me[5].kp8Config.colorOn2[0] := 'off';
   stations.me[5].kp8Config.colorOn2[4] := 'off';
   stations.me[5].kp8Config.colorOff[0] := 'off';
   stations.me[5].kp8Config.colorOff[1] := 'green';
   stations.me[5].kp8Config.colorOff[2] := 'green';
   stations.me[5].kp8Config.colorOff[3] := 'green';
   stations.me[5].kp8Config.colorOff[4] := 'off';
   stations.me[5].kp8Config.colorOff[5] := 'green';
   stations.me[5].kp8Config.colorOff[6] := 'green';
   stations.me[5].kp8Config.colorOff[7] := 'green';
   stations.me[5].kp8Config.mode[1] := TRUE;
   stations.me[5].kp8Config.mode[2] := TRUE;
   stations.me[5].kp8Config.mode[3] := TRUE;
   stations.me[5].kp8Config.mode[5] := TRUE;
   stations.me[5].kp8Config.mode[6] := TRUE;
   stations.me[5].kp8Config.mode[7] := TRUE;
   stations.me[5].kp8Out := 16#00EE_0000;
   stations.me[5].presetTime.allotted[1] := 1800.0;
   stations.me[5].presetTime.allotted[2] := 1800.0;
   stations.me[5].presetTime.allotted[3] := 1800.0;
   stations.me[5].presetTime.allotted[5] := 1800.0;
   stations.me[5].presetTime.allotted[6] := 1800.0;
   stations.me[5].presetTime.allotted[7] := 1800.0;
   stations.me[5].presetTime.critical[1] := 300.0;
   stations.me[5].presetTime.critical[2] := 300.0;
   stations.me[5].presetTime.critical[3] := 300.0;
   stations.me[5].presetTime.critical[5] := 300.0;
   stations.me[5].presetTime.critical[6] := 300.0;
   stations.me[5].presetTime.critical[7] := 300.0;
   stations.me[5].stackLightOut := 16#2449_0200;
   stations.me[6].kp8Config.activate[1] := TRUE;
   stations.me[6].kp8Config.activate[2] := TRUE;
   stations.me[6].kp8Config.activate[3] := TRUE;
   stations.me[6].kp8Config.activate[5] := TRUE;
   stations.me[6].kp8Config.activate[6] := TRUE;
   stations.me[6].kp8Config.activate[7] := TRUE;
   stations.me[6].kp8Config.colorOn1[0] := 'off';
   stations.me[6].kp8Config.colorOn1[1] := 'yellow';
   stations.me[6].kp8Config.colorOn1[2] := 'yellow';
   stations.me[6].kp8Config.colorOn1[3] := 'yellow';
   stations.me[6].kp8Config.colorOn1[4] := 'off';
   stations.me[6].kp8Config.colorOn1[5] := 'yellow';
   stations.me[6].kp8Config.colorOn1[6] := 'yellow';
   stations.me[6].kp8Config.colorOn1[7] := 'yellow';
   stations.me[6].kp8Config.colorOn2[0] := 'off';
   stations.me[6].kp8Config.colorOn2[4] := 'off';
   stations.me[6].kp8Config.colorOff[0] := 'off';
   stations.me[6].kp8Config.colorOff[1] := 'green';
   stations.me[6].kp8Config.colorOff[2] := 'green';
   stations.me[6].kp8Config.colorOff[3] := 'green';
   stations.me[6].kp8Config.colorOff[4] := 'off';
   stations.me[6].kp8Config.colorOff[5] := 'green';
   stations.me[6].kp8Config.colorOff[6] := 'green';
   stations.me[6].kp8Config.colorOff[7] := 'green';
   stations.me[6].kp8Config.mode[1] := TRUE;
   stations.me[6].kp8Config.mode[2] := TRUE;
   stations.me[6].kp8Config.mode[3] := TRUE;
   stations.me[6].kp8Config.mode[5] := TRUE;
   stations.me[6].kp8Config.mode[6] := TRUE;
   stations.me[6].kp8Config.mode[7] := TRUE;
   stations.me[6].kp8Out := 16#00EE_0000;
   stations.me[6].presetTime.allotted[1] := 1800.0;
   stations.me[6].presetTime.allotted[2] := 1800.0;
   stations.me[6].presetTime.allotted[3] := 1800.0;
   stations.me[6].presetTime.allotted[5] := 1800.0;
   stations.me[6].presetTime.allotted[6] := 1800.0;
   stations.me[6].presetTime.allotted[7] := 1800.0;
   stations.me[6].presetTime.critical[1] := 300.0;
   stations.me[6].presetTime.critical[2] := 300.0;
   stations.me[6].presetTime.critical[3] := 300.0;
   stations.me[6].presetTime.critical[5] := 300.0;
   stations.me[6].presetTime.critical[6] := 300.0;
   stations.me[6].presetTime.critical[7] := 300.0;
   stations.me[6].stackLightOut := 16#2449_0200;
   stations.me[7].kp8Config.activate[3] := TRUE;
   stations.me[7].kp8Config.activate[6] := TRUE;
   stations.me[7].kp8Config.activate[7] := TRUE;
   stations.me[7].kp8Config.colorOn1[0] := 'off';
   stations.me[7].kp8Config.colorOn1[1] := 'off';
   stations.me[7].kp8Config.colorOn1[2] := 'off';
   stations.me[7].kp8Config.colorOn1[3] := 'yellow';
   stations.me[7].kp8Config.colorOn1[4] := 'off';
   stations.me[7].kp8Config.colorOn1[5] := 'off';
   stations.me[7].kp8Config.colorOn1[6] := 'yellow';
   stations.me[7].kp8Config.colorOn1[7] := 'yellow';
   stations.me[7].kp8Config.colorOn2[0] := 'off';
   stations.me[7].kp8Config.colorOn2[1] := 'off';
   stations.me[7].kp8Config.colorOn2[2] := 'off';
   stations.me[7].kp8Config.colorOn2[4] := 'off';
   stations.me[7].kp8Config.colorOn2[5] := 'off';
   stations.me[7].kp8Config.colorOff[0] := 'off';
   stations.me[7].kp8Config.colorOff[1] := 'off';
   stations.me[7].kp8Config.colorOff[2] := 'off';
   stations.me[7].kp8Config.colorOff[3] := 'green';
   stations.me[7].kp8Config.colorOff[4] := 'off';
   stations.me[7].kp8Config.colorOff[5] := 'off';
   stations.me[7].kp8Config.colorOff[6] := 'green';
   stations.me[7].kp8Config.colorOff[7] := 'green';
   stations.me[7].kp8Config.mode[3] := TRUE;
   stations.me[7].kp8Config.mode[6] := TRUE;
   stations.me[7].kp8Config.mode[7] := TRUE;
   stations.me[7].kp8Out := 16#00C8_0000;
   stations.me[7].presetTime.allotted[3] := 1800.0;
   stations.me[7].presetTime.allotted[6] := 1800.0;
   stations.me[7].presetTime.allotted[7] := 1800.0;
   stations.me[7].presetTime.critical[3] := 300.0;
   stations.me[7].presetTime.critical[6] := 300.0;
   stations.me[7].presetTime.critical[7] := 300.0;
   stations.me[7].settings.btnSelection[3] := TRUE;
   stations.me[7].stackLightOut := 16#2401_0000;
   stations.me[8].kp8Config.activate[3] := TRUE;
   stations.me[8].kp8Config.activate[6] := TRUE;
   stations.me[8].kp8Config.activate[7] := TRUE;
   stations.me[8].kp8Config.colorOn1[0] := 'off';
   stations.me[8].kp8Config.colorOn1[1] := 'off';
   stations.me[8].kp8Config.colorOn1[2] := 'off';
   stations.me[8].kp8Config.colorOn1[3] := 'yellow';
   stations.me[8].kp8Config.colorOn1[4] := 'off';
   stations.me[8].kp8Config.colorOn1[5] := 'off';
   stations.me[8].kp8Config.colorOn1[6] := 'yellow';
   stations.me[8].kp8Config.colorOn1[7] := 'yellow';
   stations.me[8].kp8Config.colorOn2[0] := 'off';
   stations.me[8].kp8Config.colorOn2[1] := 'off';
   stations.me[8].kp8Config.colorOn2[2] := 'off';
   stations.me[8].kp8Config.colorOn2[4] := 'off';
   stations.me[8].kp8Config.colorOn2[5] := 'off';
   stations.me[8].kp8Config.colorOff[0] := 'off';
   stations.me[8].kp8Config.colorOff[1] := 'off';
   stations.me[8].kp8Config.colorOff[2] := 'off';
   stations.me[8].kp8Config.colorOff[3] := 'green';
   stations.me[8].kp8Config.colorOff[4] := 'off';
   stations.me[8].kp8Config.colorOff[5] := 'off';
   stations.me[8].kp8Config.colorOff[6] := 'green';
   stations.me[8].kp8Config.colorOff[7] := 'green';
   stations.me[8].kp8Config.mode[3] := TRUE;
   stations.me[8].kp8Config.mode[6] := TRUE;
   stations.me[8].kp8Config.mode[7] := TRUE;
   stations.me[8].kp8Out := 16#00C8_0000;
   stations.me[8].presetTime.allotted[3] := 1800.0;
   stations.me[8].presetTime.allotted[6] := 1800.0;
   stations.me[8].presetTime.allotted[7] := 1800.0;
   stations.me[8].presetTime.critical[3] := 300.0;
   stations.me[8].presetTime.critical[6] := 300.0;
   stations.me[8].presetTime.critical[7] := 300.0;
   stations.me[8].stackLightOut := 16#2401_0000;
   stations.me[9].kp8Config.activate[3] := TRUE;
   stations.me[9].kp8Config.activate[7] := TRUE;
   stations.me[9].kp8Config.colorOn1[0] := 'off';
   stations.me[9].kp8Config.colorOn1[1] := 'off';
   stations.me[9].kp8Config.colorOn1[2] := 'off';
   stations.me[9].kp8Config.colorOn1[3] := 'yellow';
   stations.me[9].kp8Config.colorOn1[4] := 'off';
   stations.me[9].kp8Config.colorOn1[5] := 'off';
   stations.me[9].kp8Config.colorOn1[6] := 'off';
   stations.me[9].kp8Config.colorOn1[7] := 'yellow';
   stations.me[9].kp8Config.colorOn2[0] := 'off';
   stations.me[9].kp8Config.colorOn2[1] := 'off';
   stations.me[9].kp8Config.colorOn2[2] := 'off';
   stations.me[9].kp8Config.colorOn2[4] := 'off';
   stations.me[9].kp8Config.colorOn2[5] := 'off';
   stations.me[9].kp8Config.colorOn2[6] := 'off';
   stations.me[9].kp8Config.colorOff[0] := 'off';
   stations.me[9].kp8Config.colorOff[1] := 'off';
   stations.me[9].kp8Config.colorOff[2] := 'off';
   stations.me[9].kp8Config.colorOff[3] := 'green';
   stations.me[9].kp8Config.colorOff[4] := 'off';
   stations.me[9].kp8Config.colorOff[5] := 'off';
   stations.me[9].kp8Config.colorOff[6] := 'off';
   stations.me[9].kp8Config.colorOff[7] := 'green';
   stations.me[9].kp8Config.mode[3] := TRUE;
   stations.me[9].kp8Config.mode[7] := TRUE;
   stations.me[9].kp8Out := 16#0088_0000;
   stations.me[9].presetTime.allotted[3] := 1800.0;
   stations.me[9].presetTime.allotted[7] := 1800.0;
   stations.me[9].presetTime.critical[3] := 300.0;
   stations.me[9].presetTime.critical[7] := 300.0;
   stations.me[9].stackLightOut := 16#2400_0000;
   stations.me[10].kp8Config.activate[3] := TRUE;
   stations.me[10].kp8Config.activate[6] := TRUE;
   stations.me[10].kp8Config.activate[7] := TRUE;
   stations.me[10].kp8Config.colorOn1[0] := 'off';
   stations.me[10].kp8Config.colorOn1[1] := 'off';
   stations.me[10].kp8Config.colorOn1[2] := 'off';
   stations.me[10].kp8Config.colorOn1[3] := 'yellow';
   stations.me[10].kp8Config.colorOn1[4] := 'off';
   stations.me[10].kp8Config.colorOn1[5] := 'off';
   stations.me[10].kp8Config.colorOn1[6] := 'yellow';
   stations.me[10].kp8Config.colorOn1[7] := 'yellow';
   stations.me[10].kp8Config.colorOn2[0] := 'off';
   stations.me[10].kp8Config.colorOn2[1] := 'off';
   stations.me[10].kp8Config.colorOn2[2] := 'off';
   stations.me[10].kp8Config.colorOn2[4] := 'off';
   stations.me[10].kp8Config.colorOn2[5] := 'off';
   stations.me[10].kp8Config.colorOff[0] := 'off';
   stations.me[10].kp8Config.colorOff[1] := 'off';
   stations.me[10].kp8Config.colorOff[2] := 'off';
   stations.me[10].kp8Config.colorOff[3] := 'green';
   stations.me[10].kp8Config.colorOff[4] := 'off';
   stations.me[10].kp8Config.colorOff[5] := 'off';
   stations.me[10].kp8Config.colorOff[6] := 'green';
   stations.me[10].kp8Config.colorOff[7] := 'green';
   stations.me[10].kp8Config.mode[3] := TRUE;
   stations.me[10].kp8Config.mode[6] := TRUE;
   stations.me[10].kp8Config.mode[7] := TRUE;
   stations.me[10].kp8Out := 16#00C8_0000;
   stations.me[10].presetTime.allotted[3] := 1800.0;
   stations.me[10].presetTime.allotted[6] := 1800.0;
   stations.me[10].presetTime.allotted[7] := 1800.0;
   stations.me[10].presetTime.critical[3] := 300.0;
   stations.me[10].presetTime.critical[6] := 300.0;
   stations.me[10].presetTime.critical[7] := 300.0;
   stations.me[10].stackLightOut := 16#2401_0000;
   stations.me[11].kp8Config.activate[3] := TRUE;
   stations.me[11].kp8Config.activate[6] := TRUE;
   stations.me[11].kp8Config.activate[7] := TRUE;
   stations.me[11].kp8Config.colorOn1[0] := 'off';
   stations.me[11].kp8Config.colorOn1[1] := 'off';
   stations.me[11].kp8Config.colorOn1[2] := 'off';
   stations.me[11].kp8Config.colorOn1[3] := 'yellow';
   stations.me[11].kp8Config.colorOn1[4] := 'off';
   stations.me[11].kp8Config.colorOn1[5] := 'off';
   stations.me[11].kp8Config.colorOn1[6] := 'yellow';
   stations.me[11].kp8Config.colorOn1[7] := 'yellow';
   stations.me[11].kp8Config.colorOn2[0] := 'off';
   stations.me[11].kp8Config.colorOn2[1] := 'off';
   stations.me[11].kp8Config.colorOn2[2] := 'off';
   stations.me[11].kp8Config.colorOn2[4] := 'off';
   stations.me[11].kp8Config.colorOn2[5] := 'off';
   stations.me[11].kp8Config.colorOff[0] := 'off';
   stations.me[11].kp8Config.colorOff[1] := 'off';
   stations.me[11].kp8Config.colorOff[2] := 'off';
   stations.me[11].kp8Config.colorOff[3] := 'green';
   stations.me[11].kp8Config.colorOff[4] := 'off';
   stations.me[11].kp8Config.colorOff[5] := 'off';
   stations.me[11].kp8Config.colorOff[6] := 'green';
   stations.me[11].kp8Config.colorOff[7] := 'green';
   stations.me[11].kp8Config.mode[3] := TRUE;
   stations.me[11].kp8Config.mode[6] := TRUE;
   stations.me[11].kp8Config.mode[7] := TRUE;
   stations.me[11].kp8Out := 16#00C8_0000;
   stations.me[11].presetTime.allotted[3] := 1800.0;
   stations.me[11].presetTime.allotted[6] := 1800.0;
   stations.me[11].presetTime.allotted[7] := 1800.0;
   stations.me[11].presetTime.critical[3] := 300.0;
   stations.me[11].presetTime.critical[6] := 300.0;
   stations.me[11].presetTime.critical[7] := 300.0;
   stations.me[11].stackLightOut := 16#2401_0000;
   stations.me[12].kp8Config.activate[1] := TRUE;
   stations.me[12].kp8Config.activate[2] := TRUE;
   stations.me[12].kp8Config.activate[3] := TRUE;
   stations.me[12].kp8Config.activate[5] := TRUE;
   stations.me[12].kp8Config.activate[6] := TRUE;
   stations.me[12].kp8Config.activate[7] := TRUE;
   stations.me[12].kp8Config.colorOn1[0] := 'off';
   stations.me[12].kp8Config.colorOn1[1] := 'yellow';
   stations.me[12].kp8Config.colorOn1[2] := 'yellow';
   stations.me[12].kp8Config.colorOn1[3] := 'yellow';
   stations.me[12].kp8Config.colorOn1[4] := 'off';
   stations.me[12].kp8Config.colorOn1[5] := 'yellow';
   stations.me[12].kp8Config.colorOn1[6] := 'yellow';
   stations.me[12].kp8Config.colorOn1[7] := 'yellow';
   stations.me[12].kp8Config.colorOn2[0] := 'off';
   stations.me[12].kp8Config.colorOn2[4] := 'off';
   stations.me[12].kp8Config.colorOff[0] := 'off';
   stations.me[12].kp8Config.colorOff[1] := 'green';
   stations.me[12].kp8Config.colorOff[2] := 'green';
   stations.me[12].kp8Config.colorOff[3] := 'green';
   stations.me[12].kp8Config.colorOff[4] := 'off';
   stations.me[12].kp8Config.colorOff[5] := 'green';
   stations.me[12].kp8Config.colorOff[6] := 'green';
   stations.me[12].kp8Config.colorOff[7] := 'green';
   stations.me[12].kp8Config.mode[1] := TRUE;
   stations.me[12].kp8Config.mode[2] := TRUE;
   stations.me[12].kp8Config.mode[3] := TRUE;
   stations.me[12].kp8Config.mode[5] := TRUE;
   stations.me[12].kp8Config.mode[6] := TRUE;
   stations.me[12].kp8Config.mode[7] := TRUE;
   stations.me[12].kp8Out := 16#00EE_0000;
   stations.me[12].presetTime.allotted[1] := 1800.0;
   stations.me[12].presetTime.allotted[2] := 1800.0;
   stations.me[12].presetTime.allotted[3] := 1800.0;
   stations.me[12].presetTime.allotted[5] := 1800.0;
   stations.me[12].presetTime.allotted[6] := 1800.0;
   stations.me[12].presetTime.allotted[7] := 1800.0;
   stations.me[12].presetTime.critical[1] := 300.0;
   stations.me[12].presetTime.critical[2] := 300.0;
   stations.me[12].presetTime.critical[3] := 300.0;
   stations.me[12].presetTime.critical[5] := 300.0;
   stations.me[12].presetTime.critical[6] := 300.0;
   stations.me[12].presetTime.critical[7] := 300.0;
   stations.me[12].stackLightOut := 16#2449_0200;
   stations.me[13].kp8Config.activate[2] := TRUE;
   stations.me[13].kp8Config.activate[3] := TRUE;
   stations.me[13].kp8Config.activate[6] := TRUE;
   stations.me[13].kp8Config.activate[7] := TRUE;
   stations.me[13].kp8Config.colorOn1[0] := 'off';
   stations.me[13].kp8Config.colorOn1[1] := 'off';
   stations.me[13].kp8Config.colorOn1[2] := 'yellow';
   stations.me[13].kp8Config.colorOn1[3] := 'yellow';
   stations.me[13].kp8Config.colorOn1[4] := 'off';
   stations.me[13].kp8Config.colorOn1[5] := 'off';
   stations.me[13].kp8Config.colorOn1[6] := 'yellow';
   stations.me[13].kp8Config.colorOn1[7] := 'yellow';
   stations.me[13].kp8Config.colorOn2[0] := 'off';
   stations.me[13].kp8Config.colorOn2[1] := 'off';
   stations.me[13].kp8Config.colorOn2[4] := 'off';
   stations.me[13].kp8Config.colorOn2[5] := 'off';
   stations.me[13].kp8Config.colorOff[0] := 'off';
   stations.me[13].kp8Config.colorOff[1] := 'off';
   stations.me[13].kp8Config.colorOff[2] := 'green';
   stations.me[13].kp8Config.colorOff[3] := 'green';
   stations.me[13].kp8Config.colorOff[4] := 'off';
   stations.me[13].kp8Config.colorOff[5] := 'off';
   stations.me[13].kp8Config.colorOff[6] := 'green';
   stations.me[13].kp8Config.colorOff[7] := 'green';
   stations.me[13].kp8Config.mode[2] := TRUE;
   stations.me[13].kp8Config.mode[3] := TRUE;
   stations.me[13].kp8Config.mode[6] := TRUE;
   stations.me[13].kp8Config.mode[7] := TRUE;
   stations.me[13].kp8Out := 16#00CC_0000;
   stations.me[13].presetTime.allotted[2] := 1800.0;
   stations.me[13].presetTime.allotted[3] := 1800.0;
   stations.me[13].presetTime.allotted[6] := 1800.0;
   stations.me[13].presetTime.allotted[7] := 1800.0;
   stations.me[13].presetTime.critical[2] := 300.0;
   stations.me[13].presetTime.critical[3] := 300.0;
   stations.me[13].presetTime.critical[6] := 300.0;
   stations.me[13].presetTime.critical[7] := 300.0;
   stations.me[13].stackLightOut := 16#2409_0000;
   stations.me[14].kp8Config.activate[2] := TRUE;
   stations.me[14].kp8Config.activate[3] := TRUE;
   stations.me[14].kp8Config.activate[5] := TRUE;
   stations.me[14].kp8Config.activate[6] := TRUE;
   stations.me[14].kp8Config.activate[7] := TRUE;
   stations.me[14].kp8Config.colorOn1[0] := 'off';
   stations.me[14].kp8Config.colorOn1[1] := 'off';
   stations.me[14].kp8Config.colorOn1[2] := 'yellow';
   stations.me[14].kp8Config.colorOn1[3] := 'yellow';
   stations.me[14].kp8Config.colorOn1[4] := 'off';
   stations.me[14].kp8Config.colorOn1[5] := 'yellow';
   stations.me[14].kp8Config.colorOn1[6] := 'yellow';
   stations.me[14].kp8Config.colorOn1[7] := 'yellow';
   stations.me[14].kp8Config.colorOn2[0] := 'off';
   stations.me[14].kp8Config.colorOn2[1] := 'off';
   stations.me[14].kp8Config.colorOn2[4] := 'off';
   stations.me[14].kp8Config.colorOff[0] := 'off';
   stations.me[14].kp8Config.colorOff[1] := 'off';
   stations.me[14].kp8Config.colorOff[2] := 'green';
   stations.me[14].kp8Config.colorOff[3] := 'green';
   stations.me[14].kp8Config.colorOff[4] := 'off';
   stations.me[14].kp8Config.colorOff[5] := 'green';
   stations.me[14].kp8Config.colorOff[6] := 'green';
   stations.me[14].kp8Config.colorOff[7] := 'green';
   stations.me[14].kp8Config.mode[2] := TRUE;
   stations.me[14].kp8Config.mode[3] := TRUE;
   stations.me[14].kp8Config.mode[5] := TRUE;
   stations.me[14].kp8Config.mode[6] := TRUE;
   stations.me[14].kp8Config.mode[7] := TRUE;
   stations.me[14].kp8Out := 16#00EC_0000;
   stations.me[14].presetTime.allotted[2] := 1800.0;
   stations.me[14].presetTime.allotted[3] := 1800.0;
   stations.me[14].presetTime.allotted[5] := 1800.0;
   stations.me[14].presetTime.allotted[6] := 1800.0;
   stations.me[14].presetTime.allotted[7] := 1800.0;
   stations.me[14].presetTime.critical[2] := 300.0;
   stations.me[14].presetTime.critical[3] := 300.0;
   stations.me[14].presetTime.critical[5] := 300.0;
   stations.me[14].presetTime.critical[6] := 300.0;
   stations.me[14].presetTime.critical[7] := 300.0;
   stations.me[14].stackLightOut := 16#2449_0000;
   stations.me[15].kp8Config.activate[1] := TRUE;
   stations.me[15].kp8Config.activate[2] := TRUE;
   stations.me[15].kp8Config.activate[3] := TRUE;
   stations.me[15].kp8Config.activate[5] := TRUE;
   stations.me[15].kp8Config.activate[6] := TRUE;
   stations.me[15].kp8Config.activate[7] := TRUE;
   stations.me[15].kp8Config.colorOn1[0] := 'off';
   stations.me[15].kp8Config.colorOn1[1] := 'yellow';
   stations.me[15].kp8Config.colorOn1[2] := 'yellow';
   stations.me[15].kp8Config.colorOn1[3] := 'yellow';
   stations.me[15].kp8Config.colorOn1[4] := 'off';
   stations.me[15].kp8Config.colorOn1[5] := 'yellow';
   stations.me[15].kp8Config.colorOn1[6] := 'yellow';
   stations.me[15].kp8Config.colorOn1[7] := 'yellow';
   stations.me[15].kp8Config.colorOn2[0] := 'off';
   stations.me[15].kp8Config.colorOn2[4] := 'off';
   stations.me[15].kp8Config.colorOff[0] := 'off';
   stations.me[15].kp8Config.colorOff[1] := 'green';
   stations.me[15].kp8Config.colorOff[2] := 'green';
   stations.me[15].kp8Config.colorOff[3] := 'green';
   stations.me[15].kp8Config.colorOff[4] := 'off';
   stations.me[15].kp8Config.colorOff[5] := 'green';
   stations.me[15].kp8Config.colorOff[6] := 'green';
   stations.me[15].kp8Config.colorOff[7] := 'green';
   stations.me[15].kp8Config.mode[1] := TRUE;
   stations.me[15].kp8Config.mode[2] := TRUE;
   stations.me[15].kp8Config.mode[3] := TRUE;
   stations.me[15].kp8Config.mode[5] := TRUE;
   stations.me[15].kp8Config.mode[6] := TRUE;
   stations.me[15].kp8Config.mode[7] := TRUE;
   stations.me[15].kp8Out := 16#00EE_0000;
   stations.me[15].presetTime.allotted[1] := 1800.0;
   stations.me[15].presetTime.allotted[2] := 1800.0;
   stations.me[15].presetTime.allotted[3] := 1800.0;
   stations.me[15].presetTime.allotted[5] := 1800.0;
   stations.me[15].presetTime.allotted[6] := 1800.0;
   stations.me[15].presetTime.allotted[7] := 1800.0;
   stations.me[15].presetTime.critical[1] := 300.0;
   stations.me[15].presetTime.critical[2] := 300.0;
   stations.me[15].presetTime.critical[3] := 300.0;
   stations.me[15].presetTime.critical[5] := 300.0;
   stations.me[15].presetTime.critical[6] := 300.0;
   stations.me[15].presetTime.critical[7] := 300.0;
   stations.me[15].stackLightOut := 16#2449_0200;
   stations.me[16].kp8Config.activate[3] := TRUE;
   stations.me[16].kp8Config.activate[7] := TRUE;
   stations.me[16].kp8Config.colorOn1[0] := 'off';
   stations.me[16].kp8Config.colorOn1[1] := 'off';
   stations.me[16].kp8Config.colorOn1[2] := 'off';
   stations.me[16].kp8Config.colorOn1[3] := 'yellow';
   stations.me[16].kp8Config.colorOn1[4] := 'off';
   stations.me[16].kp8Config.colorOn1[5] := 'off';
   stations.me[16].kp8Config.colorOn1[6] := 'off';
   stations.me[16].kp8Config.colorOn1[7] := 'yellow';
   stations.me[16].kp8Config.colorOn2[0] := 'off';
   stations.me[16].kp8Config.colorOn2[1] := 'off';
   stations.me[16].kp8Config.colorOn2[2] := 'off';
   stations.me[16].kp8Config.colorOn2[4] := 'off';
   stations.me[16].kp8Config.colorOn2[5] := 'off';
   stations.me[16].kp8Config.colorOn2[6] := 'off';
   stations.me[16].kp8Config.colorOff[0] := 'off';
   stations.me[16].kp8Config.colorOff[1] := 'off';
   stations.me[16].kp8Config.colorOff[2] := 'off';
   stations.me[16].kp8Config.colorOff[3] := 'green';
   stations.me[16].kp8Config.colorOff[4] := 'off';
   stations.me[16].kp8Config.colorOff[5] := 'off';
   stations.me[16].kp8Config.colorOff[6] := 'off';
   stations.me[16].kp8Config.colorOff[7] := 'green';
   stations.me[16].kp8Config.mode[3] := TRUE;
   stations.me[16].kp8Config.mode[7] := TRUE;
   stations.me[16].kp8Out := 16#0088_0000;
   stations.me[16].presetTime.allotted[3] := 1800.0;
   stations.me[16].presetTime.allotted[6] := 1800.0;
   stations.me[16].presetTime.allotted[7] := 1800.0;
   stations.me[16].presetTime.critical[3] := 300.0;
   stations.me[16].presetTime.critical[6] := 300.0;
   stations.me[16].presetTime.critical[7] := 300.0;
   stations.me[16].stackLightOut := 16#2400_0000;
   stations.me[17].kp8Config.activate[2] := TRUE;
   stations.me[17].kp8Config.activate[3] := TRUE;
   stations.me[17].kp8Config.activate[6] := TRUE;
   stations.me[17].kp8Config.activate[7] := TRUE;
   stations.me[17].kp8Config.colorOn1[0] := 'off';
   stations.me[17].kp8Config.colorOn1[1] := 'off';
   stations.me[17].kp8Config.colorOn1[2] := 'yellow';
   stations.me[17].kp8Config.colorOn1[3] := 'yellow';
   stations.me[17].kp8Config.colorOn1[4] := 'off';
   stations.me[17].kp8Config.colorOn1[5] := 'off';
   stations.me[17].kp8Config.colorOn1[6] := 'yellow';
   stations.me[17].kp8Config.colorOn1[7] := 'yellow';
   stations.me[17].kp8Config.colorOn2[0] := 'off';
   stations.me[17].kp8Config.colorOn2[1] := 'off';
   stations.me[17].kp8Config.colorOn2[4] := 'off';
   stations.me[17].kp8Config.colorOn2[5] := 'off';
   stations.me[17].kp8Config.colorOff[0] := 'off';
   stations.me[17].kp8Config.colorOff[1] := 'off';
   stations.me[17].kp8Config.colorOff[2] := 'green';
   stations.me[17].kp8Config.colorOff[3] := 'green';
   stations.me[17].kp8Config.colorOff[4] := 'off';
   stations.me[17].kp8Config.colorOff[5] := 'off';
   stations.me[17].kp8Config.colorOff[6] := 'green';
   stations.me[17].kp8Config.colorOff[7] := 'green';
   stations.me[17].kp8Config.mode[2] := TRUE;
   stations.me[17].kp8Config.mode[3] := TRUE;
   stations.me[17].kp8Config.mode[6] := TRUE;
   stations.me[17].kp8Config.mode[7] := TRUE;
   stations.me[17].kp8Out := 16#00CC_0000;
   stations.me[17].presetTime.allotted[2] := 1800.0;
   stations.me[17].presetTime.allotted[3] := 1800.0;
   stations.me[17].presetTime.allotted[6] := 1800.0;
   stations.me[17].presetTime.allotted[7] := 1800.0;
   stations.me[17].presetTime.critical[2] := 300.0;
   stations.me[17].presetTime.critical[3] := 300.0;
   stations.me[17].presetTime.critical[6] := 300.0;
   stations.me[17].presetTime.critical[7] := 300.0;
   stations.me[17].stackLightOut := 16#2409_0000;
   stations.me[18].kp8Config.activate[3] := TRUE;
   stations.me[18].kp8Config.activate[6] := TRUE;
   stations.me[18].kp8Config.activate[7] := TRUE;
   stations.me[18].kp8Config.colorOn1[0] := 'off';
   stations.me[18].kp8Config.colorOn1[1] := 'off';
   stations.me[18].kp8Config.colorOn1[2] := 'off';
   stations.me[18].kp8Config.colorOn1[3] := 'yellow';
   stations.me[18].kp8Config.colorOn1[4] := 'off';
   stations.me[18].kp8Config.colorOn1[5] := 'off';
   stations.me[18].kp8Config.colorOn1[6] := 'yellow';
   stations.me[18].kp8Config.colorOn1[7] := 'yellow';
   stations.me[18].kp8Config.colorOn2[0] := 'off';
   stations.me[18].kp8Config.colorOn2[1] := 'off';
   stations.me[18].kp8Config.colorOn2[2] := 'off';
   stations.me[18].kp8Config.colorOn2[4] := 'off';
   stations.me[18].kp8Config.colorOn2[5] := 'off';
   stations.me[18].kp8Config.colorOff[0] := 'off';
   stations.me[18].kp8Config.colorOff[1] := 'off';
   stations.me[18].kp8Config.colorOff[2] := 'off';
   stations.me[18].kp8Config.colorOff[3] := 'green';
   stations.me[18].kp8Config.colorOff[4] := 'off';
   stations.me[18].kp8Config.colorOff[5] := 'off';
   stations.me[18].kp8Config.colorOff[6] := 'green';
   stations.me[18].kp8Config.colorOff[7] := 'green';
   stations.me[18].kp8Config.mode[3] := TRUE;
   stations.me[18].kp8Config.mode[6] := TRUE;
   stations.me[18].kp8Config.mode[7] := TRUE;
   stations.me[18].kp8Out := 16#00C8_0000;
   stations.me[18].presetTime.allotted[3] := 1800.0;
   stations.me[18].presetTime.allotted[6] := 1800.0;
   stations.me[18].presetTime.allotted[7] := 1800.0;
   stations.me[18].presetTime.critical[3] := 300.0;
   stations.me[18].presetTime.critical[6] := 300.0;
   stations.me[18].presetTime.critical[7] := 300.0;
   stations.me[18].stackLightOut := 16#2401_0000;
   stations.me[19].kp8Config.activate[1] := TRUE;
   stations.me[19].kp8Config.activate[2] := TRUE;
   stations.me[19].kp8Config.activate[3] := TRUE;
   stations.me[19].kp8Config.activate[5] := TRUE;
   stations.me[19].kp8Config.activate[6] := TRUE;
   stations.me[19].kp8Config.activate[7] := TRUE;
   stations.me[19].kp8Config.colorOn1[0] := 'off';
   stations.me[19].kp8Config.colorOn1[1] := 'yellow';
   stations.me[19].kp8Config.colorOn1[2] := 'yellow';
   stations.me[19].kp8Config.colorOn1[3] := 'yellow';
   stations.me[19].kp8Config.colorOn1[4] := 'off';
   stations.me[19].kp8Config.colorOn1[5] := 'yellow';
   stations.me[19].kp8Config.colorOn1[6] := 'yellow';
   stations.me[19].kp8Config.colorOn1[7] := 'yellow';
   stations.me[19].kp8Config.colorOn2[0] := 'off';
   stations.me[19].kp8Config.colorOn2[4] := 'off';
   stations.me[19].kp8Config.colorOff[0] := 'off';
   stations.me[19].kp8Config.colorOff[1] := 'green';
   stations.me[19].kp8Config.colorOff[2] := 'green';
   stations.me[19].kp8Config.colorOff[3] := 'green';
   stations.me[19].kp8Config.colorOff[4] := 'off';
   stations.me[19].kp8Config.colorOff[5] := 'green';
   stations.me[19].kp8Config.colorOff[6] := 'green';
   stations.me[19].kp8Config.colorOff[7] := 'green';
   stations.me[19].kp8Config.mode[1] := TRUE;
   stations.me[19].kp8Config.mode[2] := TRUE;
   stations.me[19].kp8Config.mode[3] := TRUE;
   stations.me[19].kp8Config.mode[5] := TRUE;
   stations.me[19].kp8Config.mode[6] := TRUE;
   stations.me[19].kp8Config.mode[7] := TRUE;
   stations.me[19].kp8Out := 16#00EE_0000;
   stations.me[19].presetTime.allotted[1] := 1800.0;
   stations.me[19].presetTime.allotted[2] := 1800.0;
   stations.me[19].presetTime.allotted[3] := 1800.0;
   stations.me[19].presetTime.allotted[5] := 120.0;
   stations.me[19].presetTime.allotted[6] := 1800.0;
   stations.me[19].presetTime.allotted[7] := 1800.0;
   stations.me[19].presetTime.critical[1] := 300.0;
   stations.me[19].presetTime.critical[2] := 300.0;
   stations.me[19].presetTime.critical[3] := 300.0;
   stations.me[19].presetTime.critical[5] := 70.0;
   stations.me[19].presetTime.critical[6] := 300.0;
   stations.me[19].presetTime.critical[7] := 300.0;
   stations.me[19].settings.selected := TRUE;
   stations.me[19].stackLightOut := 16#2449_0200;
   stations.me[20].kp8Config.colorOn1[0] := 'off';
   stations.me[20].kp8Config.colorOn1[1] := 'off';
   stations.me[20].kp8Config.colorOn1[2] := 'off';
   stations.me[20].kp8Config.colorOn1[3] := 'off';
   stations.me[20].kp8Config.colorOn1[4] := 'off';
   stations.me[20].kp8Config.colorOn1[5] := 'off';
   stations.me[20].kp8Config.colorOn1[6] := 'off';
   stations.me[20].kp8Config.colorOn1[7] := 'off';
   stations.me[20].kp8Config.colorOn2[0] := 'off';
   stations.me[20].kp8Config.colorOn2[1] := 'off';
   stations.me[20].kp8Config.colorOn2[2] := 'off';
   stations.me[20].kp8Config.colorOn2[3] := 'off';
   stations.me[20].kp8Config.colorOn2[4] := 'off';
   stations.me[20].kp8Config.colorOn2[5] := 'off';
   stations.me[20].kp8Config.colorOn2[6] := 'off';
   stations.me[20].kp8Config.colorOn2[7] := 'off';
   stations.me[20].kp8Config.colorOff[0] := 'off';
   stations.me[20].kp8Config.colorOff[1] := 'off';
   stations.me[20].kp8Config.colorOff[2] := 'off';
   stations.me[20].kp8Config.colorOff[3] := 'off';
   stations.me[20].kp8Config.colorOff[4] := 'off';
   stations.me[20].kp8Config.colorOff[5] := 'off';
   stations.me[20].kp8Config.colorOff[6] := 'off';
   stations.me[20].kp8Config.colorOff[7] := 'off';
   stations.me[20].kp8Out := 16#0000_0000;
   stations.me[20].stackLightOut := 16#0000_0000;
   stations.me[21].kp8Config.activate[7] := TRUE;
   stations.me[21].kp8Config.colorOn1[0] := 'off';
   stations.me[21].kp8Config.colorOn1[1] := 'off';
   stations.me[21].kp8Config.colorOn1[2] := 'off';
   stations.me[21].kp8Config.colorOn1[3] := 'off';
   stations.me[21].kp8Config.colorOn1[4] := 'off';
   stations.me[21].kp8Config.colorOn1[5] := 'off';
   stations.me[21].kp8Config.colorOn1[6] := 'off';
   stations.me[21].kp8Config.colorOn1[7] := 'yellow';
   stations.me[21].kp8Config.colorOn2[0] := 'off';
   stations.me[21].kp8Config.colorOn2[1] := 'off';
   stations.me[21].kp8Config.colorOn2[2] := 'off';
   stations.me[21].kp8Config.colorOn2[3] := 'off';
   stations.me[21].kp8Config.colorOn2[4] := 'off';
   stations.me[21].kp8Config.colorOn2[5] := 'off';
   stations.me[21].kp8Config.colorOn2[6] := 'off';
   stations.me[21].kp8Config.colorOff[0] := 'off';
   stations.me[21].kp8Config.colorOff[1] := 'off';
   stations.me[21].kp8Config.colorOff[2] := 'off';
   stations.me[21].kp8Config.colorOff[3] := 'off';
   stations.me[21].kp8Config.colorOff[4] := 'off';
   stations.me[21].kp8Config.colorOff[5] := 'off';
   stations.me[21].kp8Config.colorOff[6] := 'off';
   stations.me[21].kp8Config.colorOff[7] := 'green';
   stations.me[21].kp8Config.mode[7] := TRUE;
   stations.me[21].kp8Out := 16#0080_0000;
   stations.me[21].presetTime.allotted[7] := 1800.0;
   stations.me[21].presetTime.critical[7] := 300.0;
   stations.me[21].stackLightOut := 16#0400_0000;
   stations.me[22].kp8Config.activate[3] := TRUE;
   stations.me[22].kp8Config.activate[6] := TRUE;
   stations.me[22].kp8Config.activate[7] := TRUE;
   stations.me[22].kp8Config.colorOn1[0] := 'off';
   stations.me[22].kp8Config.colorOn1[1] := 'off';
   stations.me[22].kp8Config.colorOn1[2] := 'off';
   stations.me[22].kp8Config.colorOn1[3] := 'yellow';
   stations.me[22].kp8Config.colorOn1[4] := 'off';
   stations.me[22].kp8Config.colorOn1[5] := 'off';
   stations.me[22].kp8Config.colorOn1[6] := 'yellow';
   stations.me[22].kp8Config.colorOn1[7] := 'yellow';
   stations.me[22].kp8Config.colorOn2[0] := 'off';
   stations.me[22].kp8Config.colorOn2[1] := 'off';
   stations.me[22].kp8Config.colorOn2[2] := 'off';
   stations.me[22].kp8Config.colorOn2[4] := 'off';
   stations.me[22].kp8Config.colorOn2[5] := 'off';
   stations.me[22].kp8Config.colorOff[0] := 'off';
   stations.me[22].kp8Config.colorOff[1] := 'off';
   stations.me[22].kp8Config.colorOff[2] := 'off';
   stations.me[22].kp8Config.colorOff[3] := 'green';
   stations.me[22].kp8Config.colorOff[4] := 'off';
   stations.me[22].kp8Config.colorOff[5] := 'off';
   stations.me[22].kp8Config.colorOff[6] := 'green';
   stations.me[22].kp8Config.colorOff[7] := 'green';
   stations.me[22].kp8Config.mode[3] := TRUE;
   stations.me[22].kp8Config.mode[6] := TRUE;
   stations.me[22].kp8Config.mode[7] := TRUE;
   stations.me[22].kp8Out := 16#00C8_0000;
   stations.me[22].presetTime.allotted[3] := 1800.0;
   stations.me[22].presetTime.allotted[6] := 1800.0;
   stations.me[22].presetTime.allotted[7] := 1800.0;
   stations.me[22].presetTime.critical[3] := 300.0;
   stations.me[22].presetTime.critical[6] := 300.0;
   stations.me[22].presetTime.critical[7] := 300.0;
   stations.me[22].stackLightOut := 16#2401_0000;
   stations.me[23].kp8Config.activate[7] := TRUE;
   stations.me[23].kp8Config.colorOn1[0] := 'off';
   stations.me[23].kp8Config.colorOn1[1] := 'off';
   stations.me[23].kp8Config.colorOn1[2] := 'off';
   stations.me[23].kp8Config.colorOn1[3] := 'off';
   stations.me[23].kp8Config.colorOn1[4] := 'off';
   stations.me[23].kp8Config.colorOn1[5] := 'off';
   stations.me[23].kp8Config.colorOn1[6] := 'off';
   stations.me[23].kp8Config.colorOn1[7] := 'yellow';
   stations.me[23].kp8Config.colorOn2[0] := 'off';
   stations.me[23].kp8Config.colorOn2[1] := 'off';
   stations.me[23].kp8Config.colorOn2[2] := 'off';
   stations.me[23].kp8Config.colorOn2[3] := 'off';
   stations.me[23].kp8Config.colorOn2[4] := 'off';
   stations.me[23].kp8Config.colorOn2[5] := 'off';
   stations.me[23].kp8Config.colorOn2[6] := 'off';
   stations.me[23].kp8Config.colorOff[0] := 'off';
   stations.me[23].kp8Config.colorOff[1] := 'off';
   stations.me[23].kp8Config.colorOff[2] := 'off';
   stations.me[23].kp8Config.colorOff[3] := 'off';
   stations.me[23].kp8Config.colorOff[4] := 'off';
   stations.me[23].kp8Config.colorOff[5] := 'off';
   stations.me[23].kp8Config.colorOff[6] := 'off';
   stations.me[23].kp8Config.colorOff[7] := 'green';
   stations.me[23].kp8Config.mode[7] := TRUE;
   stations.me[23].kp8Out := 16#0080_0000;
   stations.me[23].presetTime.allotted[7] := 1800.0;
   stations.me[23].presetTime.critical[7] := 300.0;
   stations.me[23].stackLightOut := 16#0400_0000;
   stations.me[24].kp8Config.activate[7] := TRUE;
   stations.me[24].kp8Config.colorOn1[0] := 'off';
   stations.me[24].kp8Config.colorOn1[1] := 'off';
   stations.me[24].kp8Config.colorOn1[2] := 'off';
   stations.me[24].kp8Config.colorOn1[3] := 'off';
   stations.me[24].kp8Config.colorOn1[4] := 'off';
   stations.me[24].kp8Config.colorOn1[5] := 'off';
   stations.me[24].kp8Config.colorOn1[6] := 'off';
   stations.me[24].kp8Config.colorOn1[7] := 'yellow';
   stations.me[24].kp8Config.colorOn2[0] := 'off';
   stations.me[24].kp8Config.colorOn2[1] := 'off';
   stations.me[24].kp8Config.colorOn2[2] := 'off';
   stations.me[24].kp8Config.colorOn2[3] := 'off';
   stations.me[24].kp8Config.colorOn2[4] := 'off';
   stations.me[24].kp8Config.colorOn2[5] := 'off';
   stations.me[24].kp8Config.colorOn2[6] := 'off';
   stations.me[24].kp8Config.colorOff[0] := 'off';
   stations.me[24].kp8Config.colorOff[1] := 'off';
   stations.me[24].kp8Config.colorOff[2] := 'off';
   stations.me[24].kp8Config.colorOff[3] := 'off';
   stations.me[24].kp8Config.colorOff[4] := 'off';
   stations.me[24].kp8Config.colorOff[5] := 'off';
   stations.me[24].kp8Config.colorOff[6] := 'off';
   stations.me[24].kp8Config.colorOff[7] := 'green';
   stations.me[24].kp8Config.mode[7] := TRUE;
   stations.me[24].kp8Out := 16#0080_0000;
   stations.me[24].partNumbers[0] := WSTRING#'';
   stations.me[24].partNumbers[1] := WSTRING#'';
   stations.me[24].partNumbers[2] := WSTRING#'';
   stations.me[24].partNumbers[3] := WSTRING#'';
   stations.me[24].partNumbers[4] := WSTRING#'';
   stations.me[24].partNumbers[5] := WSTRING#'';
   stations.me[24].partNumbers[6] := WSTRING#'';
   stations.me[24].presetTime.allotted[7] := 1800.0;
   stations.me[24].presetTime.critical[7] := 300.0;
   stations.me[24].stackLightOut := 16#0400_0000;
   stations.me[25].btnStates[0] := TRUE;
   stations.me[25].kp8Config.activate[1] := TRUE;
   stations.me[25].kp8Config.activate[2] := TRUE;
   stations.me[25].kp8Config.activate[6] := TRUE;
   stations.me[25].kp8Config.activate[7] := TRUE;
   stations.me[25].kp8Config.colorOn1[0] := 'off';
   stations.me[25].kp8Config.colorOn1[1] := 'yellow';
   stations.me[25].kp8Config.colorOn1[2] := 'yellow';
   stations.me[25].kp8Config.colorOn1[3] := 'off';
   stations.me[25].kp8Config.colorOn1[4] := 'off';
   stations.me[25].kp8Config.colorOn1[5] := 'off';
   stations.me[25].kp8Config.colorOn1[6] := 'yellow';
   stations.me[25].kp8Config.colorOn1[7] := 'yellow';
   stations.me[25].kp8Config.colorOn2[0] := 'off';
   stations.me[25].kp8Config.colorOn2[3] := 'off';
   stations.me[25].kp8Config.colorOn2[4] := 'off';
   stations.me[25].kp8Config.colorOn2[5] := 'off';
   stations.me[25].kp8Config.colorOff[0] := 'off';
   stations.me[25].kp8Config.colorOff[1] := 'green';
   stations.me[25].kp8Config.colorOff[2] := 'green';
   stations.me[25].kp8Config.colorOff[3] := 'off';
   stations.me[25].kp8Config.colorOff[4] := 'off';
   stations.me[25].kp8Config.colorOff[5] := 'off';
   stations.me[25].kp8Config.colorOff[6] := 'green';
   stations.me[25].kp8Config.colorOff[7] := 'green';
   stations.me[25].kp8Config.mode[1] := TRUE;
   stations.me[25].kp8Config.mode[2] := TRUE;
   stations.me[25].kp8Config.mode[6] := TRUE;
   stations.me[25].kp8Config.mode[7] := TRUE;
   stations.me[25].kp8Out := 16#4000_8400;
   stations.me[25].partNumbers[0] := WSTRING#'';
   stations.me[25].partNumbers[1] := WSTRING#'C/O MATERIALS';
   stations.me[25].partNumbers[2] := WSTRING#'16.08.216.806.020A';
   stations.me[25].partNumbers[3] := WSTRING#'';
   stations.me[25].partNumbers[4] := WSTRING#'';
   stations.me[25].partNumbers[5] := WSTRING#'';
   stations.me[25].partNumbers[6] := WSTRING#'16.08.208.631.000F';
   stations.me[25].partNumbers[7] := WSTRING#'16.08.216.315.000A';
   stations.me[25].presetTime.allotted[1] := 1800.0;
   stations.me[25].presetTime.allotted[2] := 1800.0;
   stations.me[25].presetTime.allotted[6] := 1800.0;
   stations.me[25].presetTime.allotted[7] := 1800.0;
   stations.me[25].presetTime.critical[1] := 300.0;
   stations.me[25].presetTime.critical[2] := 300.0;
   stations.me[25].presetTime.critical[6] := 300.0;
   stations.me[25].presetTime.critical[7] := 300.0;
   stations.me[25].settings.btnSelection[1] := TRUE;
   stations.me[25].stackLightOut := 16#0409_0200;
   stations.me[26].animations[3] := 3;
   stations.me[26].btnStates[3] := TRUE;
   stations.me[26].elapsedTime.partReq[3] := 2305.576;
   stations.me[26].kp8Config.activate[1] := TRUE;
   stations.me[26].kp8Config.activate[2] := TRUE;
   stations.me[26].kp8Config.activate[3] := TRUE;
   stations.me[26].kp8Config.activate[5] := TRUE;
   stations.me[26].kp8Config.activate[6] := TRUE;
   stations.me[26].kp8Config.activate[7] := TRUE;
   stations.me[26].kp8Config.colorOn1[0] := 'off';
   stations.me[26].kp8Config.colorOn1[1] := 'yellow';
   stations.me[26].kp8Config.colorOn1[2] := 'yellow';
   stations.me[26].kp8Config.colorOn1[3] := 'yellow';
   stations.me[26].kp8Config.colorOn1[4] := 'off';
   stations.me[26].kp8Config.colorOn1[5] := 'yellow';
   stations.me[26].kp8Config.colorOn1[6] := 'yellow';
   stations.me[26].kp8Config.colorOn1[7] := 'yellow';
   stations.me[26].kp8Config.colorOn2[0] := 'off';
   stations.me[26].kp8Config.colorOn2[4] := 'off';
   stations.me[26].kp8Config.colorOff[0] := 'off';
   stations.me[26].kp8Config.colorOff[1] := 'green';
   stations.me[26].kp8Config.colorOff[2] := 'green';
   stations.me[26].kp8Config.colorOff[3] := 'green';
   stations.me[26].kp8Config.colorOff[4] := 'off';
   stations.me[26].kp8Config.colorOff[5] := 'green';
   stations.me[26].kp8Config.colorOff[6] := 'green';
   stations.me[26].kp8Config.colorOff[7] := 'green';
   stations.me[26].kp8Config.mode[1] := TRUE;
   stations.me[26].kp8Config.mode[2] := TRUE;
   stations.me[26].kp8Config.mode[3] := TRUE;
   stations.me[26].kp8Config.mode[5] := TRUE;
   stations.me[26].kp8Config.mode[6] := TRUE;
   stations.me[26].kp8Config.mode[7] := TRUE;
   stations.me[26].kp8Out := 16#E000_0000;
   stations.me[26].partNumbers[0] := WSTRING#'';
   stations.me[26].partNumbers[1] := WSTRING#'C/O MATERIALS';
   stations.me[26].partNumbers[2] := WSTRING#'16.08.216.291.000A';
   stations.me[26].partNumbers[3] := WSTRING#'16.08.216.315.001A';
   stations.me[26].partNumbers[4] := WSTRING#'';
   stations.me[26].partNumbers[5] := WSTRING#'16.08.216.057.001A';
   stations.me[26].partNumbers[6] := WSTRING#'16.08.208.661.000F';
   stations.me[26].partNumbers[7] := WSTRING#'16.08.216.315.002A';
   stations.me[26].partOrdered[3] := TRUE;
   stations.me[26].partRequested[3] := TRUE;
   stations.me[26].presetTime.allotted[1] := 1800.0;
   stations.me[26].presetTime.allotted[2] := 1800.0;
   stations.me[26].presetTime.allotted[3] := 1800.0;
   stations.me[26].presetTime.allotted[5] := 1800.0;
   stations.me[26].presetTime.allotted[6] := 1800.0;
   stations.me[26].presetTime.allotted[7] := 1800.0;
   stations.me[26].presetTime.critical[1] := 300.0;
   stations.me[26].presetTime.critical[2] := 300.0;
   stations.me[26].presetTime.critical[3] := 300.0;
   stations.me[26].presetTime.critical[5] := 300.0;
   stations.me[26].presetTime.critical[6] := 300.0;
   stations.me[26].presetTime.critical[7] := 300.0;
   stations.me[26].stackLightOut := 16#0449_0200;
   stations.me[27].kp8Config.activate[1] := TRUE;
   stations.me[27].kp8Config.activate[2] := TRUE;
   stations.me[27].kp8Config.activate[3] := TRUE;
   stations.me[27].kp8Config.activate[5] := TRUE;
   stations.me[27].kp8Config.activate[6] := TRUE;
   stations.me[27].kp8Config.activate[7] := TRUE;
   stations.me[27].kp8Config.colorOn1[0] := 'off';
   stations.me[27].kp8Config.colorOn1[1] := 'yellow';
   stations.me[27].kp8Config.colorOn1[2] := 'yellow';
   stations.me[27].kp8Config.colorOn1[3] := 'yellow';
   stations.me[27].kp8Config.colorOn1[4] := 'off';
   stations.me[27].kp8Config.colorOn1[5] := 'yellow';
   stations.me[27].kp8Config.colorOn1[6] := 'yellow';
   stations.me[27].kp8Config.colorOn1[7] := 'yellow';
   stations.me[27].kp8Config.colorOn2[0] := 'off';
   stations.me[27].kp8Config.colorOn2[4] := 'off';
   stations.me[27].kp8Config.colorOff[0] := 'off';
   stations.me[27].kp8Config.colorOff[1] := 'green';
   stations.me[27].kp8Config.colorOff[2] := 'green';
   stations.me[27].kp8Config.colorOff[3] := 'green';
   stations.me[27].kp8Config.colorOff[4] := 'off';
   stations.me[27].kp8Config.colorOff[5] := 'green';
   stations.me[27].kp8Config.colorOff[6] := 'green';
   stations.me[27].kp8Config.colorOff[7] := 'green';
   stations.me[27].kp8Config.mode[1] := TRUE;
   stations.me[27].kp8Config.mode[2] := TRUE;
   stations.me[27].kp8Config.mode[3] := TRUE;
   stations.me[27].kp8Config.mode[5] := TRUE;
   stations.me[27].kp8Config.mode[6] := TRUE;
   stations.me[27].kp8Config.mode[7] := TRUE;
   stations.me[27].kp8Out := 16#4000_A800;
   stations.me[27].partNumbers[0] := WSTRING#'';
   stations.me[27].partNumbers[1] := WSTRING#'C/O MATERIALS';
   stations.me[27].partNumbers[2] := WSTRING#'16.18.011.301.010A';
   stations.me[27].partNumbers[3] := WSTRING#'16.18.011.301.020B';
   stations.me[27].partNumbers[4] := WSTRING#'';
   stations.me[27].partNumbers[5] := WSTRING#'16.18.007.311.010A';
   stations.me[27].partNumbers[6] := WSTRING#'16.18.007.311.020A';
   stations.me[27].partNumbers[7] := WSTRING#'16.18.012.401.020A';
   stations.me[27].presetTime.allotted[1] := 1800.0;
   stations.me[27].presetTime.allotted[2] := 1800.0;
   stations.me[27].presetTime.allotted[3] := 1800.0;
   stations.me[27].presetTime.allotted[5] := 1800.0;
   stations.me[27].presetTime.allotted[6] := 1800.0;
   stations.me[27].presetTime.allotted[7] := 1800.0;
   stations.me[27].presetTime.critical[1] := 300.0;
   stations.me[27].presetTime.critical[2] := 300.0;
   stations.me[27].presetTime.critical[3] := 300.0;
   stations.me[27].presetTime.critical[5] := 300.0;
   stations.me[27].presetTime.critical[6] := 300.0;
   stations.me[27].presetTime.critical[7] := 300.0;
   stations.me[27].stackLightOut := 16#2449_0200;
   stations.me[28].kp8Config.activate[1] := TRUE;
   stations.me[28].kp8Config.activate[3] := TRUE;
   stations.me[28].kp8Config.activate[6] := TRUE;
   stations.me[28].kp8Config.activate[7] := TRUE;
   stations.me[28].kp8Config.colorOn1[0] := 'off';
   stations.me[28].kp8Config.colorOn1[1] := 'yellow';
   stations.me[28].kp8Config.colorOn1[2] := 'off';
   stations.me[28].kp8Config.colorOn1[3] := 'yellow';
   stations.me[28].kp8Config.colorOn1[4] := 'off';
   stations.me[28].kp8Config.colorOn1[5] := 'off';
   stations.me[28].kp8Config.colorOn1[6] := 'yellow';
   stations.me[28].kp8Config.colorOn1[7] := 'yellow';
   stations.me[28].kp8Config.colorOn2[0] := 'off';
   stations.me[28].kp8Config.colorOn2[2] := 'off';
   stations.me[28].kp8Config.colorOn2[4] := 'off';
   stations.me[28].kp8Config.colorOn2[5] := 'off';
   stations.me[28].kp8Config.colorOff[0] := 'off';
   stations.me[28].kp8Config.colorOff[1] := 'green';
   stations.me[28].kp8Config.colorOff[2] := 'off';
   stations.me[28].kp8Config.colorOff[3] := 'green';
   stations.me[28].kp8Config.colorOff[4] := 'off';
   stations.me[28].kp8Config.colorOff[5] := 'off';
   stations.me[28].kp8Config.colorOff[6] := 'green';
   stations.me[28].kp8Config.colorOff[7] := 'green';
   stations.me[28].kp8Config.mode[1] := TRUE;
   stations.me[28].kp8Config.mode[3] := TRUE;
   stations.me[28].kp8Config.mode[6] := TRUE;
   stations.me[28].kp8Config.mode[7] := TRUE;
   stations.me[28].kp8Out := 16#0000_6E00;
   stations.me[28].partNumbers[0] := WSTRING#'';
   stations.me[28].partNumbers[1] := WSTRING#'C/O MATERIALS';
   stations.me[28].partNumbers[2] := WSTRING#'';
   stations.me[28].partNumbers[3] := WSTRING#'16.32.112.543.210E';
   stations.me[28].partNumbers[4] := WSTRING#'';
   stations.me[28].partNumbers[5] := WSTRING#'';
   stations.me[28].partNumbers[6] := WSTRING#'16.32.112.543.020A';
   stations.me[28].partNumbers[7] := WSTRING#'16.32.112.315.018A';
   stations.me[28].presetTime.allotted[1] := 1800.0;
   stations.me[28].presetTime.allotted[3] := 1800.0;
   stations.me[28].presetTime.allotted[6] := 1800.0;
   stations.me[28].presetTime.allotted[7] := 1800.0;
   stations.me[28].presetTime.critical[1] := 300.0;
   stations.me[28].presetTime.critical[3] := 300.0;
   stations.me[28].presetTime.critical[6] := 300.0;
   stations.me[28].presetTime.critical[7] := 300.0;
   stations.me[28].stackLightOut := 16#2401_0200;
   stations.me[29].kp8Config.activate[1] := TRUE;
   stations.me[29].kp8Config.activate[2] := TRUE;
   stations.me[29].kp8Config.activate[3] := TRUE;
   stations.me[29].kp8Config.activate[5] := TRUE;
   stations.me[29].kp8Config.activate[6] := TRUE;
   stations.me[29].kp8Config.activate[7] := TRUE;
   stations.me[29].kp8Config.colorOn1[0] := 'off';
   stations.me[29].kp8Config.colorOn1[1] := 'yellow';
   stations.me[29].kp8Config.colorOn1[2] := 'yellow';
   stations.me[29].kp8Config.colorOn1[3] := 'yellow';
   stations.me[29].kp8Config.colorOn1[4] := 'off';
   stations.me[29].kp8Config.colorOn1[5] := 'yellow';
   stations.me[29].kp8Config.colorOn1[6] := 'yellow';
   stations.me[29].kp8Config.colorOn1[7] := 'yellow';
   stations.me[29].kp8Config.colorOn2[0] := 'off';
   stations.me[29].kp8Config.colorOn2[4] := 'off';
   stations.me[29].kp8Config.colorOff[0] := 'off';
   stations.me[29].kp8Config.colorOff[1] := 'green';
   stations.me[29].kp8Config.colorOff[2] := 'green';
   stations.me[29].kp8Config.colorOff[3] := 'green';
   stations.me[29].kp8Config.colorOff[4] := 'off';
   stations.me[29].kp8Config.colorOff[5] := 'green';
   stations.me[29].kp8Config.colorOff[6] := 'green';
   stations.me[29].kp8Config.colorOff[7] := 'green';
   stations.me[29].kp8Config.mode[1] := TRUE;
   stations.me[29].kp8Config.mode[2] := TRUE;
   stations.me[29].kp8Config.mode[3] := TRUE;
   stations.me[29].kp8Config.mode[5] := TRUE;
   stations.me[29].kp8Config.mode[6] := TRUE;
   stations.me[29].kp8Config.mode[7] := TRUE;
   stations.me[29].kp8Out := 16#2A00_4400;
   stations.me[29].partNumbers[0] := WSTRING#'';
   stations.me[29].partNumbers[1] := WSTRING#'C/O MATERIALS';
   stations.me[29].partNumbers[2] := WSTRING#'11.54.007.052.007B';
   stations.me[29].partNumbers[3] := WSTRING#'11.54.007.315.026G';
   stations.me[29].partNumbers[4] := WSTRING#'';
   stations.me[29].partNumbers[5] := WSTRING#'11.54.007.052.008A';
   stations.me[29].partNumbers[6] := WSTRING#'11.54.007.045.015D';
   stations.me[29].partNumbers[7] := WSTRING#'11.54.017.315.001F';
   stations.me[29].presetTime.allotted[1] := 1800.0;
   stations.me[29].presetTime.allotted[2] := 1800.0;
   stations.me[29].presetTime.allotted[3] := 1800.0;
   stations.me[29].presetTime.allotted[5] := 1800.0;
   stations.me[29].presetTime.allotted[6] := 1800.0;
   stations.me[29].presetTime.allotted[7] := 1800.0;
   stations.me[29].presetTime.critical[1] := 300.0;
   stations.me[29].presetTime.critical[2] := 300.0;
   stations.me[29].presetTime.critical[3] := 300.0;
   stations.me[29].presetTime.critical[5] := 300.0;
   stations.me[29].presetTime.critical[6] := 300.0;
   stations.me[29].presetTime.critical[7] := 300.0;
   stations.me[29].settings.btnSelection[3] := TRUE;
   stations.me[29].stackLightOut := 16#2449_0200;
   stations.me[30].kp8Config.activate[7] := TRUE;
   stations.me[30].kp8Config.colorOn1[0] := 'off';
   stations.me[30].kp8Config.colorOn1[1] := 'off';
   stations.me[30].kp8Config.colorOn1[2] := 'off';
   stations.me[30].kp8Config.colorOn1[3] := 'off';
   stations.me[30].kp8Config.colorOn1[4] := 'off';
   stations.me[30].kp8Config.colorOn1[5] := 'off';
   stations.me[30].kp8Config.colorOn1[6] := 'off';
   stations.me[30].kp8Config.colorOn1[7] := 'yellow';
   stations.me[30].kp8Config.colorOn2[0] := 'off';
   stations.me[30].kp8Config.colorOn2[1] := 'off';
   stations.me[30].kp8Config.colorOn2[2] := 'off';
   stations.me[30].kp8Config.colorOn2[3] := 'off';
   stations.me[30].kp8Config.colorOn2[4] := 'off';
   stations.me[30].kp8Config.colorOn2[5] := 'off';
   stations.me[30].kp8Config.colorOn2[6] := 'off';
   stations.me[30].kp8Config.colorOff[0] := 'off';
   stations.me[30].kp8Config.colorOff[1] := 'off';
   stations.me[30].kp8Config.colorOff[2] := 'off';
   stations.me[30].kp8Config.colorOff[3] := 'off';
   stations.me[30].kp8Config.colorOff[4] := 'off';
   stations.me[30].kp8Config.colorOff[5] := 'off';
   stations.me[30].kp8Config.colorOff[6] := 'off';
   stations.me[30].kp8Config.colorOff[7] := 'green';
   stations.me[30].kp8Config.mode[7] := TRUE;
   stations.me[30].kp8Out := 16#0080_0000;
   stations.me[30].partNumbers[0] := WSTRING#'';
   stations.me[30].partNumbers[1] := WSTRING#'';
   stations.me[30].partNumbers[2] := WSTRING#'';
   stations.me[30].partNumbers[3] := WSTRING#'';
   stations.me[30].partNumbers[4] := WSTRING#'';
   stations.me[30].partNumbers[5] := WSTRING#'';
   stations.me[30].partNumbers[6] := WSTRING#'';
   stations.me[30].presetTime.allotted[7] := 1800.0;
   stations.me[30].presetTime.critical[7] := 300.0;
   stations.me[30].settings.btnSelection[7] := TRUE;
   stations.me[30].stackLightOut := 16#0400_0000;
   stations.me[31].kp8Config.activate[3] := TRUE;
   stations.me[31].kp8Config.activate[7] := TRUE;
   stations.me[31].kp8Config.colorOn1[0] := 'off';
   stations.me[31].kp8Config.colorOn1[1] := 'off';
   stations.me[31].kp8Config.colorOn1[2] := 'off';
   stations.me[31].kp8Config.colorOn1[3] := 'yellow';
   stations.me[31].kp8Config.colorOn1[4] := 'off';
   stations.me[31].kp8Config.colorOn1[5] := 'off';
   stations.me[31].kp8Config.colorOn1[6] := 'off';
   stations.me[31].kp8Config.colorOn1[7] := 'yellow';
